(* IEC 61131-3 sources: F100R_S278_Temperville/MyController.device.xml.v3^/Plc Logic.plclogic.xml.v3^/Application.application.xml.v3^, 20 files *)

(* ---- GVL_Alarmes.gvl ---- *)
VAR_GLOBAL
	AlmMotor: ARRAY[1..25] OF BOOL;
	AlmValvAberta: ARRAY[1..12] OF BOOL;
	AlmValvFechada: ARRAY[1..12] OF BOOL;
	AlmGeral: ARRAY[1..12] OF BOOL;
	AlmEncoder: ARRAY[1..12] OF BOOL;
	AlmMotorParado: ARRAY[1..25] OF BOOL;
	xAlarmeSsrSuperiorAberto: ARRAY[1..60] OF BOOL;
	xAlarmeSsrSuperiorFechado: ARRAY[1..60] OF BOOL;
	xAlarmeSsrInferiorAberto: ARRAY[1..60] OF BOOL;
	xAlarmeSsrInferiorFechado: ARRAY[1..60] OF BOOL;
	xAlarmeResistRompidaSuperior: ARRAY[1..60] OF BOOL;
	xAlarmeResistRompidaInferior: ARRAY[1..60] OF BOOL;
	xAlarmeResistForceInferior: ARRAY[1..60] OF BOOL;
	xAlarmeResistForceSuperior: ARRAY[1..60] OF BOOL;
	xFalhaForcadaInferior: ARRAY[1..60] OF BOOL;
	xFalhaForcadaSuperior: ARRAY[1..60] OF BOOL;
	xAlarmesTestesResistenciasInferiores: ARRAY[1..60] OF BOOL;
	xAlarmesTestesResistenciasSuperiores: ARRAY[1..60] OF BOOL;
	AlmTermoparAbertoSuperior: ARRAY[1..60] OF BOOL;
	AlmTermoparAbertoInferior: ARRAY[1..60] OF BOOL;
	AlmTemperaturaExcedeuSuperior: ARRAY[1..60] OF BOOL;
	AlmTemperaturaExcedeuInferior: ARRAY[1..60] OF BOOL;
	xAlarmeSsr01ConvecEntAberto: BOOL;
	xAlarmeSsr01ConvecEntFechado: BOOL;
	xAlarmeSsr02ConvecEntAberto: BOOL;
	xAlarmeSsr02ConvecEntFechado: BOOL;
	xAlarmeSsr03ConvecEntAberto: BOOL;
	xAlarmeSsr03ConvecEntFechado: BOOL;
	xAlarmeSsr01ConvecSaiAberto: BOOL;
	xAlarmeSsr01ConvecSaiFechado: BOOL;
	xAlarmeSsr02ConvecSaiAberto: BOOL;
	xAlarmeSsr02ConvecSaiFechado: BOOL;
	xAlarmeSsr03ConvecSaiAberto: BOOL;
	xAlarmeSsr03ConvecSaiFechado: BOOL;
END_VAR

(* ---- GVL_ClpSuper.gvl ---- *)
VAR_GLOBAL
	/// LEITURA
	///Parâmetros On-line
	sEntradaNomedaReceita: STRING;
	sFornoNomedaReceita: STRING;
	sResfriamentoNomedaReceita: STRING;
	iEntradaEspessuraVidro: INT;
	iFornoEspessuraVidro: INT;
	iResfriamentoEspessuraVidro: INT;
	xEntradaReenvioRec: BOOL;
	xFornoReenvioRec: BOOL;
	xResfriamentoReenvioRec: BOOL;
	xPassagemReenvioRec: BOOL;
	rTemperaturaInferiorAtual: ARRAY[1..50] OF REAL;
	rTemperaturaSuperiorAtual: ARRAY[1..50] OF REAL;
	iTemperaturaPainel: INT;
	rMediaLogiaTempInferior: REAL;
	rMediaLogiaTempSuperior: REAL;
	rMediaLogicaTemperaturaTotal: REAL;
	iTempoDelayCargaDecorrido: INT;
	iTempoPausaRoleteDecorrido: INT;
	iTempoPausaRoleteRestante: INT;
	iTempoAquecFornoDecorrido: INT;
	iTempoAquecFornoRestante: INT;
	iTempoTrocaVelocidadeDecorrido: INT;
	///////////////////
	iTempoTrocaPosicaoDecorrido: INT;
	//////////////////
	iTempoTesteNobreak: TON;
	iTempoTesteNobreakRestante: INT;
	iTempoPausaResistInfDecorrido: INT;
	iTempoPausaResistSupDecorrido: INT;
	iTempoPausa02ResistSupDecorrido: INT;
	iTempoParaInicioPausaDecor: INT;
	iTempoConveccaoDecorrido: INT;
	iTempoResfriamentoDecorrido: INT;
	iTempoResfriamentoRestante: INT;
	iTempoTrocaEstagioDecorrido: INT;
	iTempoTrocaEstagio02Decorrido: INT;
	iAlturaAtualDuctosResfriadorInf01: INT;
	iAlturaAtualDuctosResfriadorSup01: INT;
	iAlturaAtualDuctosResfriadorInf02: INT;
	iAlturaAtualDuctosResfriadorSup02: INT;
	iAlturaAtualGuilhotina01: INT;
	iAlturaAtualGuilhotina01Sup: INT;
	iAlturaAtualGuilhotina01Inf: INT;
	iAlturaAtualGuilhotina02: INT;
	rTemperaturaPirometroInferior: REAL;
	rTemperaturaPirometroSuperior: REAL;
	iTempoStdByTemperDecorrido: INT;
	iTempoPassoSemEnerg	: INT ;
	rValorPressaoRedeMpa: REAL;
	rValorPressaoRedeBar: REAL;
	rValorPressaoRedePsi: REAL;
	///Polegada de Mercurio
	rValorPressaoRedeInHg: REAL;
	///Centimetro de Mercurio
	rValorPressaoRedeCmHg: REAL;
	///Milimetro de Mercurio
	rValorPressaoRedeMmHg: REAL;
	///Milimetro de Coluna d´agua
	rValorPressaoRedeMmCa: REAL;
	rValorPressaoMaqMpa: REAL;
	rValorPressaoMaqBar: REAL;
	rValorPressaoMaqPsi: REAL;
	///Polegada de Mercurio
	rValorPressaoMaqInHg: REAL;
	///Centimetro de Mercurio
	rValorPressaoMaqCmHg: REAL;
	///Milimetro de Mercurio
	rValorPressaoMaqMmHg: REAL;
	///Milimetro de Coluna d´agua
	rValorPressaoMaqMmCa: REAL;
	rTemperaturaTermocamera: REAL;
	rTemperaturaConveccaoEnt: REAL;
	rTemperaturaConveccaoSai: REAL;
	rValorLeituraPressaoDifusor01MBar: REAL;
	rValorLeituraPressaoDifusor01Bar: REAL;
	rValorLeituraPressaoDifusor01Psi: REAL;
	///Polegada de Mercurio
	rValorLeituraPressaoDifusor01InHg: REAL;
	///Centimetro de Mercurio
	rValorLeituraPressaoDifusor01CmHg: REAL;
	///Milimetro de Mercurio
	rValorLeituraPressaoDifusor01MmHg: REAL;
	///Milimetro de Coluna d´agua
	rValorLeituraPressaoDifusor01MmCa: REAL;
	rValorLeituraPressaoDifusor02MBar: REAL;
	rValorLeituraPressaoDifusor02Bar: REAL;
	rValorLeituraPressaoDifusor02Psi: REAL;
	///Polegada de Mercurio
	rValorLeituraPressaoDifusor02InHg: REAL;
	///Centimetro de Mercurio
	rValorLeituraPressaoDifusor02CmHg: REAL;
	///Milimetro de Mercurio
	rValorLeituraPressaoDifusor02MmHg: REAL;
	///Milimetro de Coluna d´agua
	rValorLeituraPressaoDifusor02MmCa: REAL;
	rValorVibracaoVent01: REAL;
	rValorVibracaoVent02: REAL;
	rValorVibracaoVent03: REAL;
	xResistenciaHabilitadaInferior: ARRAY[1..50] OF BOOL;
	xResistenciaHabilitadaSuperior: ARRAY[1..50] OF BOOL;
	xResistenciaHabilitada: ARRAY[1..50] OF BOOL;
	xResistenciaForcadaInferior: ARRAY[1..50] OF BOOL;
	xResistenciaForcadaSuperior: ARRAY[1..50] OF BOOL;
	xForceLigConvecEntVent: BOOL;
	xForceLigConvecSaiVent: BOOL;
	xGeralResistenciaForcada: BOOL;
	xTesteResistencias: BOOL;
	xTesteResistenciaAutomatico: BOOL;
	xTesteResistenciaManual: BOOL;
	xTesteEntradaSaidas: BOOL;
	xSelecaoTermopares: BOOL;
	xPortaEntradaFornoForce: BOOL;
	xPortaSaidaFornoForce: BOOL;
	xForceConveccao: BOOL;
	xConveccaoHabilitado: BOOL;
	xSubindoForno: BOOL;
	xDescendoForno: BOOL;
	xLigaVentiPainelManual: BOOL;
	xStdByTemperaturaHabilitado: BOOL;
	xStdByTemperaturaDesabilit: BOOL;
	xHabDesabResistConveccaoEnt: BOOL;
	xHabDesabResistConveccaoSai: BOOL;
	xAqueceRampaPatamar: BOOL;
	xAqueceReceita: BOOL;
	xAqueceRapido: BOOL;
	xAqueceLento: BOOL;
	xFimAquecimento: BOOL;
	xDuctosInf01CheckOk: BOOL;
	xDuctosSup01CheckOk: BOOL;
	xDuctosInf02CheckOk: BOOL;
	xDuctosSup02CheckOk: BOOL;
	xGuilhotina01CheckOk: BOOL;
	xGuilhotina01SupCheckOk: BOOL;
	xGuilhotina01InfCheckOk: BOOL;
	xGuilhotina02CheckOk: BOOL;
	xDuctosInf01Enable: BOOL;
	xDuctosSup01Enable: BOOL;
	xDuctosInf02Enable: BOOL;
	xDuctosSup02Enable: BOOL;
	xGuilhotina01Enable: BOOL;
	xGuilhotina01SupEnable: BOOL;
	xGuilhotina01InfEnable: BOOL;
	xGuilhotina02Enable: BOOL;
	xEnergiaOk: BOOL;
	xSemEnergia: BOOL;
	xbRestart: BOOL;
	xTesteNobreakOK: BOOL;
	xIniciaTesteNobreak: BOOL;
	xResistenciaInferiorOn: BOOL;
	xResistenciaSuperiorOn: BOOL;
	xTesteResistenciasIniciado: BOOL;
	xFimTesteResistencias: BOOL;

	xImgSetTempStandByCiclo: BOOL;

	xCircuitoEmergenciaCC : BOOL;
	xAlertaPosChCircCC	: BOOL ;
	xHabDesabCircuitoCC	: BOOL ;

	ValorAmperagemResistenciaInferior: ARRAY[1..50] OF REAL;
	ValorAmperagemResistenciaSuperior: ARRAY[1..50] OF REAL;
	xTestandoResistenciaInferior: ARRAY[1..50] OF BOOL;
	xTestandoResistenciaSuperior: ARRAY[1..50] OF BOOL;
	xFaseReleInferior: ARRAY[1..50] OF STRING;
	xFaseReleSuperior: ARRAY[1..50] OF STRING;
	iAnimaResistenciaInferior: ARRAY[1..50] OF INT;
	iAnimaResistenciaSuperior: ARRAY[1..50] OF INT;
	iAnimaResistenciaSsr01ConvecEnt: INT;
	iAnimaResistenciaSsr02ConvecEnt: INT;
	iAnimaResistenciaSsr03ConvecEnt: INT;
	iAnimaResistenciaSsr01ConvecSai: INT;
	iAnimaResistenciaSsr02ConvecSai: INT;
	iAnimaResistenciaSsr03ConvecSai: INT;
	iAnimaStatusTesteResistencias: INT;
	iAnimaTesteResistenciaInferior: ARRAY[1..50] OF INT;
	iAnimaTesteResistenciaSuperior: ARRAY[1..50] OF INT;
	iAnimaAlarmesMotores: ARRAY[1..25] OF INT;
	iAnimaAlarmesValvulas: ARRAY[1..12] OF INT;
	xTemperaturaInfeirorOk: ARRAY[1..50] OF BOOL;
	xTemperaturaSupeirorOk: ARRAY[1..50] OF BOOL;
	///Numero de cargas que sairam do resfriamento por dia
	iContaCargasResfriamento: INT;
	/// Tags Relatório de Produção
	xIniciaRelatorioProd: BOOL;
	xFinalizaRelatorioProd: BOOL;
	uNumeroCargaRel: UINT;
	rConsumoCargaRel: REAL;
	rConsumoAquecRel: REAL;
	rConsumoDiario: REAL;
	rConsumoDiarioRel: REAL;
	xGrvRelatorioEnerg: BOOL;
	iTamanhoCargaRel: INT;
	/// Tags acerta relógio
	xAcertaRelogio: BOOL;
	xRelogioAcertado: BOOL;
	/// Relatório Aquecimento
	xIniciaRelatorioAquecRampa: BOOL;
	xFinalizaRelatorioAquecRampa: BOOL;
	xIniciaRelatorioAquecRec: BOOL;
	xFinalizaRelatorioAquecRec: BOOL;
	///Tags lógica incremento
	rIncrementoTemperSup: INT;
	rIncrementoTemperInf: INT;
	rIncrementoPotenciaSup: INT;
	rIncrementoPotenciaInf: INT;
	///Tags rampas
	rTempoRampa01: REAL;
	rTempoRampa02: REAL;
	rTempoRampa03: REAL;
END_VAR

(* ---- GVL_Encoder.gvl ---- *)
VAR_GLOBAL
	dValorEncoderForno: DINT;
	dValorEncoderResfriador: DINT;
	dValorEncoderDuctosResfriadorInf01: DINT;
	dValorEncoderDuctosResfriadorSup01: DINT;
	dValorEncoderDuctosResfriadorInf02: DINT;
	dValorEncoderDuctosResfriadorSup02: DINT;
	dValorEncoderGuilhotinaResfriador01: DINT;
	dValorEncoderGuilhotinaResfriador02: DINT;

	dValorEncoderGuilhotinaResfriador01Inf: DINT;
	dValorEncoderGuilhotinaResfriador01Sup: DINT;

	xHomeEncoderForno: BOOL;
	xHomeEncoderResfriador: BOOL;
	xHomeEncoderDuctosResfriadorInf01: BOOL;
	xHomeEncoderDuctosResfriadorSup01: BOOL;
	xHomeEncoderDuctosResfriadorInf02: BOOL;
	xHomeEncoderDuctosResfriadorSup02: BOOL;
	xHomeEncoderGuilhotinaResfriador01: BOOL;
	xHomeEncoderGuilhotinaResfriador02: BOOL;
	xHomeEncoderGuilhotinaResfriador01Sup: BOOL;
	xHomeEncoderGuilhotinaResfriador01Inf: BOOL;

	xEncoderFornoOk: BOOL;
	xEncoderResfriadorOk: BOOL;
	xEncoderDuctosResfriadorInf01Ok: BOOL;
	xEncoderDuctosResfriadorSup01Ok: BOOL;
	xEncoderDuctosResfriadorInf02Ok: BOOL;
	xEncoderDuctosResfriadorSup02Ok: BOOL;
	xEncoderGuilhotinaResfriador01Ok: BOOL;
	xEncoderGuilhotinaResfriador02Ok: BOOL;
END_VAR

(* ---- GVL_Energia.gvl ---- *)
VAR_GLOBAL
	///Parametros de leituras Instantaneas Reais do PM710 para o Supervisório
	rConsumoEnergiaReal_kWh: REAL;
	rConsumoEnergiaAparente_kVAh: REAL;
	rConsumoEnergiaReativa_kVARh: REAL;
	rPotenciaTotalReal_kW: REAL;
	rPotenciaTotalAparente_kVA: REAL;
	rPotenciaTotalReativa_kVAR: REAL;
	rFatorDePotenciaTotal: REAL;
	rTensaoFFMedia_V: REAL;
	rTensaoFNMedia_V: REAL;
	rCorrenteMedia_V: REAL;
	rFrequencia_Hz: REAL;
	rDemandaTotalReal_kW: REAL;
	rDemandaTotalAparente_kVA: REAL;
	rDemandaTotalReativa_kVAR: REAL;
	rDemandaMaximaReal_kW: REAL;
	rDemandaMaximaAparente_kVA: REAL;
	rDemandaMaximaReativa_kVAR: REAL;
	rCorrenteInstantFaseA_Amp: REAL;
	rCorrenteInstantFaseB_Amp: REAL;
	rCorrenteInstantFaseC_Amp: REAL;
	rCorrenteInstantNeutro_Amp: REAL;
	rCorrenteDemandaFaseA_Amp: REAL;
	rCorrenteDemandaFaseB_Amp: REAL;
	rCorrenteDemandaFaseC_Amp: REAL;
	rCorrenteMaximaDemandaFaseA_Amp: REAL;
	rCorrenteMaximaDemandaFaseB_Amp: REAL;
	rCorrenteMaximaDemandaFaseC_Amp: REAL;
	rTensaoFaseAB_V: REAL;
	rTensaoFaseBC_V: REAL;
	rTensaoFaseAC_V: REAL;
	rTensaoFaseAN_V: REAL;
	rTensaoFaseBN_V: REAL;
	rTensaoFaseCN_V: REAL;
	rPotenciaRealFaseA_kW: REAL;
	rPotenciaRealFaseB_kW: REAL;
	rPotenciaRealFaseC_kW: REAL;
	rPotenciaAparenteFaseA_kVA: REAL;
	rPotenciaAparenteFaseB_kVA: REAL;
	rPotenciaAparenteFaseC_kVA: REAL;
	rPotenciaReativaFaseA_kVAR: REAL;
	rPotenciaReativaFaseB_kVAR: REAL;
	rPotenciaReativaFaseC_kVAR: REAL;
	rCorrenteTHDFaseA: REAL;
	rCorrenteTHDFaseB: REAL;
	rCorrenteTHDFaseC: REAL;
	rCorrenteTHDNeutro: REAL;
	rTensaoTHDFaseAN: REAL;
	rTensaoTHDFaseBN: REAL;
	rTensaoTHDFaseCN: REAL;
	rTensaoTHDFaseAB: REAL;
	rTensaoTHDFaseBC: REAL;
	rTensaoTHDFaseAC: REAL;
	/// Valores minimos
	rPotenciaTotalRealMinima_kW: REAL;
	rPotenciaTotalAparenteMinima_kVA: REAL;
	rPotenciaTotalReativaMinima_kVAR: REAL;
	rFatorDePotenciaTotalMinima: REAL;
	rFrequenciaMinima_Hz: REAL;
	rCorrenteMinimaFaseA_Amp: REAL;
	rCorrenteMinimaFaseB_Amp: REAL;
	rCorrenteMinimaFaseC_Amp: REAL;
	rCorrenteMinimaNeutro_Amp: REAL;
	rTensaoMinimaFaseAN_V: REAL;
	rTensaoMinimaFaseBN_V: REAL;
	rTensaoMinimaFaseCN_V: REAL;
	rTensaoMinimaFaseAB_V: REAL;
	rTensaoMinimaFaseBC_V: REAL;
	rTensaoMinimaFaseAC_V: REAL;
	rCorrenteTHDMinimoFaseA: REAL;
	rCorrenteTHDMinimoFaseB: REAL;
	rCorrenteTHDMinimoFaseC: REAL;
	rCorrenteTHDMinimoNeutro: REAL;
	rTensaoTHDMinimoFaseAN: REAL;
	rTensaoTHDMinimoFaseBN: REAL;
	rTensaoTHDMinimoFaseCN: REAL;
	rTensaoTHDMinimoFaseAB: REAL;
	rTensaoTHDMinimoFaseBC: REAL;
	rTensaoTHDMinimoFaseAC: REAL;
	/// Valores Maximos
	rPotenciaTotalRealMaximo_kW: REAL;
	rPotenciaTotalAparenteMaximo_kVA: REAL;
	rPotenciaTotalReativaMaximo_kVAR: REAL;
	rFatorDePotenciaTotalMaximo: REAL;
	rFrequenciaMaxima_Hz: REAL;
	rCorrenteMaximoFaseA_Amp: REAL;
	rCorrenteMaximoFaseB_Amp: REAL;
	rCorrenteMaximoFaseC_Amp: REAL;
	rCorrenteMaximoNeutro_Amp: REAL;
	rTensaoMaximoFaseAN_V: REAL;
	rTensaoMaximoFaseBN_V: REAL;
	rTensaoMaximoFaseCN_V: REAL;
	rTensaoMaximoFaseAB_V: REAL;
	rTensaoMaximoFaseBC_V: REAL;
	rTensaoMaximoFaseAC_V: REAL;
	rCorrenteTHDMaximoFaseA: REAL;
	rCorrenteTHDMaximoFaseB: REAL;
	rCorrenteTHDMaximoFaseC: REAL;
	rCorrenteTHDMaximoNeutro: REAL;
	rTensaoTHDMaximoFaseAN: REAL;
	rTensaoTHDMaximoFaseBN: REAL;
	rTensaoTHDMaximoFaseCN: REAL;
	rTensaoTHDMaximoFaseAB: REAL;
	rTensaoTHDMaximoFaseBC: REAL;
	rTensaoTHDMaximoFaseAC: REAL;
	/// // // // // // // // //
	uMesFatura: UINT;
	uAnoFatura: UINT;
	bZeraAcumulado: BOOL;
	xCmdResetGeralPm: BOOL;
	// // // // // // // // //

END_VAR

(* ---- GVL_EntradasSaidas.gvl ---- *)
VAR_GLOBAL
	///ENTRADAS LÓGICAS
	///Encoder
	InputEncoderA_MeFor: BOOL;
	InputEncoderB_MeFor: BOOL;
	InputEncoderA_MeRes: BOOL;
	InputEncoderB_MeRes: BOOL;
	InputEncoderA_DuResSup01: BOOL;
	InputEncoderB_DuResSup01: BOOL;
	InputEncoderA_DuResInf01: BOOL;
	InputEncoderB_DuResInf01: BOOL;
	InputEncoderA_DuResSup02: BOOL;
	InputEncoderB_DuResSup02: BOOL;
	InputEncoderA_DuResInf02: BOOL;
	InputEncoderB_DuResInf02: BOOL;
	InputEncoderA_GuiRes01: BOOL;
	InputEncoderB_GuiRes01: BOOL;
	InputEncoderA_GuiRes02: BOOL;
	InputEncoderB_GuiRes02: BOOL;
	dValorEncoderFornoEntrada: DINT;
	dValorEncoderResfrEntrada: DINT;
	dValorEncoderDuctosResfrSup01Entrada: DINT;
	dValorEncoderDuctosResfrInf01Entrada: DINT;
	dValorEncoderDuctosResfrSup02Entrada: DINT;
	dValorEncoderDuctosResfrInf02Entrada: DINT;
	dValorEncoderGuilhoResfr01Entrada: DINT;
	dValorEncoderGuilhoResfr02Entrada: DINT;

	dValorEncoderGuilhoResfr01SupEntrada: DINT;
	dValorEncoderGuilhoResfr01InfEntrada: DINT;

	// Segurança Motor CC

	xChCircuitoEmergenciaCC	: BOOL ;
	xChHabDesabCircuitoCC	: BOOL ;

/// Mesa de Controle
	xBtIniciaCiclo: BOOL;
	xBtFinalizaCiclo: BOOL;
	xBtCalaAlarme: BOOL;
	xBtEmergencia: BOOL;
	xChAutomaticoManual: BOOL;
	///xChStandByOperacao:BOOL;
	xBtReinicia: BOOL;
	xBt01Emergencia: BOOL;
	xBt02Emergencia: BOOL;
	xBt03Emergencia: BOOL;
	xBt04Emergencia: BOOL;
	xBt05Emergencia: BOOL;
	xBt06Emergencia: BOOL;
	xBt07Emergencia: BOOL;
	xBt08Emergencia: BOOL;
	xBt09Emergencia: BOOL;
	xBt10Emergencia: BOOL;
	xBt01CalaAlarme: BOOL;
	xBt02CalaAlarme: BOOL;
	xReleSeguranca: BOOL;
	xQgeralMotores: BOOL;
	///Mesa de Entrada
	xSensorEntrada: BOOL;
	xSensorEntrada01: BOOL;
	xSensorEntrada02: BOOL;
	xSensorEntrada03: BOOL;
	xSensorEntrada04: BOOL;
	xSensorEntrada05: BOOL;
	xSensorEntrada06: BOOL;
	xSensorEntrada07: BOOL;
	xSensorEntrada08: BOOL;
	xSensorEntrada09: BOOL;
	xSensorEntrada10: BOOL;
	xBtHabilitaCarregamento: BOOL;
	xChAvancaMesaEntrada: BOOL;
	xChRecuaMesaEntrada: BOOL;
	xBtGradeEntrada: BOOL;
	xSensorGradeEntradaUp: BOOL;
	xSensorGradeEntradaDown: BOOL;
	xMotorEntradaOn: BOOL;
	///Basculante
	xBtAvancMesaBascul: BOOL;
	xBtRecuoMesaBascul: BOOL;
	xS01PistPneumRecuado: BOOL;
	xS02PistPneumAvancad: BOOL;
	xS03PistHidraulRecuado: BOOL;
	xS04PistHidraulAvancad: BOOL;
	xS05NivelaSubida: BOOL;
	xS06NivelaDescida: BOOL;
	///Mesa do Forno
	xSensorPortaEntrada: BOOL;
	xSensorPortaEntradaAberta: BOOL;
	xSensorPortaEntradaFechada: BOOL;
	xSensorPortaSaida: BOOL;
	xSensorPortaSaidaAberta: BOOL;
	xSensorPortaSaidaFechada: BOOL;
	xFcSegCalco01: BOOL;
	xFcSegCalco02: BOOL;
	xFcSegCalco03: BOOL;
	xFcSegCalco04: BOOL;
	xFcAbertoCaixaForno: BOOL;
	xFcFechadoCaixaForno: BOOL;
	xMotorFornoOn: BOOL;

	//Ventilador Passagem
	xResetVentilador01 : BOOL;
	xRefUpVentiladorPassagem : BOOL;
	xRefDownVentiladorPassagem : BOOL;
	//Guilhotina Passagem Inferior
	xFcMaximoGuiPassagemInf : BOOL;
	xFcMinimoGuiPassagemInf : BOOL;
	//Guilhotina Passagem Superior
	xFcMaximoGuiPassagemSup : BOOL;
	xFcMinimoGuiPassagemSup : BOOL;

	///Mesa do Resfriador
	xFcLimMaxLimpaResfriador02: BOOL;
	xFcLimMinLimpaResfriador02: BOOL;
	xChAvancoLimpaResfriador02: BOOL;
	xChRecuoLimpaResfriador02: BOOL;
	xMotorResfriadorOn: BOOL;
	///Mesa de Saída
	xChAvancaMesaSaida: BOOL;
	xChRecuaMesaSaida: BOOL;
	xSensorDesligaMesaSaida: BOOL;
	xBtGradeSaida: BOOL;
	xSensorGradeSaidaUp: BOOL;
	xSensorGradeSaidaDown: BOOL;
	xMotorSaidaOn: BOOL;
	///Resfriador Inferior 01
	xSensorAbertoResfriadorInf01: BOOL;
	xSensorFechadoResfriadorInf01: BOOL;
	xSensorEncoderResfriadorInf01: BOOL;
	xChAbreDuctosResfriadorInf01: BOOL;
	xFcMinimoSegResfriadorInf01: BOOL;
	xFcMaximoSegResfriadorInf01: BOOL;
	///Resfriador Superior 01
	xSensorAbertoResfriadorSup01: BOOL;
	xSensorFechadoResfriadorSup01: BOOL;
	xSensorEncoderResfriadorSup01: BOOL;
	xChAbreDuctosResfriadorSup01: BOOL;
	xFcMinimoSegResfriadorSup01: BOOL;
	xFcMaximoSegResfriadorSup01: BOOL;
	xValvulaVeneziana: BOOL;
	xMotorResfridorSup01Abre: BOOL;
	xMotorResfridorSup01Fecha: BOOL;
	///Resfriador Inferior 02
	xSensorAbertoResfriadorInf02: BOOL;
	xSensorFechadoResfriadorInf02: BOOL;
	xSensorEncoderResfriadorInf02: BOOL;
	xChAbreDuctosResfriadorInf02: BOOL;
	xFcMinimoSegResfriadorInf02: BOOL;
	xFcMaximoSegResfriadorInf02: BOOL;
	xMotorResfridorInf02Abre: BOOL;
	xMotorResfridorInf02Fecha: BOOL;
	///Resfriador Superior 02
	xSensorAbertoResfriadorSup02: BOOL;
	xSensorFechadoResfriadorSup02: BOOL;
	xSensorEncoderResfriadorSup02: BOOL;
	xChAbreDuctosResfriadorSup02: BOOL;
	xFcMinimoSegResfriadorSup02: BOOL;
	xFcMaximoSegResfriadorSup02: BOOL;
	xMotorResfridorSup02Abre: BOOL;
	xMotorResfridorSup02Fecha: BOOL;
	///Guilhotina 01
	xSensorPositivoGuilhotina01: BOOL;
	xSensorZeroGuilhotina01: BOOL;
	xSensorNegativoGuilhotina01: BOOL;
	xSensorEncoderGuilhotina01: BOOL;
	xMotorGuilhotina01Sobe: BOOL;
	xMotorGuilhotina01Desce: BOOL;

	xSensorAbertoGuilhotina01Sup: BOOL;
	xSensorFechadoGuilhotina01Sup: BOOL;
	xMotorGuilhotina01SupAbre: BOOL;
	xMotorGuilhotina01SupFecha: BOOL;

	xSensorAbertoGuilhotina01Inf: BOOL;
	xSensorFechadoGuilhotina01Inf: BOOL;
	xMotorGuilhotina01InfAbre: BOOL;
	xMotorGuilhotina01InfFecha: BOOL;

	///Guilhotina 02
	xSensorPositivoGuilhotina02: BOOL;
	xSensorZeroGuilhotina02: BOOL;
	xSensorNegativoGuilhotina02: BOOL;
	xSensorEncoderGuilhotina02: BOOL;
	xMotorGuilhotina02Sobe: BOOL;
	xMotorGuilhotina02Desce: BOOL;
	/// Retorno Reles Estado Sólido
	xRetornoSsrInferior: ARRAY[1..60] OF BOOL;
	xRetornoSsrSuperior: ARRAY[1..60] OF BOOL;
	xRetornoSsr01ConveccaoEnt: BOOL;
	xRetornoSsr02ConveccaoEnt: BOOL;
	xRetornoSsr03ConveccaoEnt: BOOL;
	xRetornoSsr01ConveccaoSai: BOOL;
	xRetornoSsr02ConveccaoSai: BOOL;
	xRetornoSsr03ConveccaoSai: BOOL;
	/// Retorno Rele Resistências Rompidas
	xResistRompidaInferior: ARRAY[1..60] OF BOOL;
	xResistRompidaSuperior: ARRAY[1..60] OF BOOL;
	/// Amperagem Resistências
	iAmperagemInferior: ARRAY[1..60] OF UINT;
	iAmperagemSuperior: ARRAY[1..60] OF UINT;
	/// Nobreak
	xSaidaNobreakOk: BOOL;
	/// Pressostato Rede Alimnetação de Ar Comprimido
	xPressaoBaixaMediaRede: BOOL;
	xPressaoMediaAltaRede: BOOL;
	/// Disjuntores
	xDisjResistOff: BOOL;
	xDisjResistOn: BOOL;
	xDisjGeralOff: BOOL;
	xDisjGeralOn: BOOL;

	/// Entradas Fisicas
	///TM262L10MESE8T - 0.1
	xM0_1_DI0: BOOL;
	xM0_1_DI1: BOOL;
	xM0_1_DI2: BOOL;
	xM0_1_DI3: BOOL;
	///TM3XHSC202 - 0.2
	xM0_2_DI0: BOOL;
	xM0_2_DI1: BOOL;
	xM0_2_DI2: BOOL;
	xM0_2_DI3: BOOL;
	xM0_2_DI4: BOOL;
	xM0_2_DI5: BOOL;
	xM0_2_DI6: BOOL;
	xM0_2_DI7: BOOL;
	xM0_2_DI8: BOOL;
	xM0_2_DI9: BOOL;
	///TM3XHSC202 - 0.3
	xM0_3_DI0: BOOL;
	xM0_3_DI1: BOOL;
	xM0_3_DI2: BOOL;
	xM0_3_DI3: BOOL;
	xM0_3_DI4: BOOL;
	xM0_3_DI5: BOOL;
	xM0_3_DI6: BOOL;
	xM0_3_DI7: BOOL;
	xM0_3_DI8: BOOL;
	xM0_3_DI9: BOOL;

	///TM3DM24K - 0.4
	xM0_4_DI0: BOOL;
	xM0_4_DI1: BOOL;
	xM0_4_DI2: BOOL;
	xM0_4_DI3: BOOL;
	xM0_4_DI4: BOOL;
	xM0_4_DI5: BOOL;
	xM0_4_DI6: BOOL;
	xM0_4_DI7: BOOL;
	xM0_4_DI8: BOOL;
	xM0_4_DI9: BOOL;
	xM0_4_DI10: BOOL;
	xM0_4_DI11: BOOL;
	xM0_4_DI12: BOOL;
	xM0_4_DI13: BOOL;
	xM0_4_DI14: BOOL;
	xM0_4_DI15: BOOL;
	xM0_4_DI16: BOOL;
	xM0_4_DI17: BOOL;
	xM0_4_DI18: BOOL;
	xM0_4_DI19: BOOL;
	xM0_4_DI20: BOOL;
	xM0_4_DI21: BOOL;
	xM0_4_DI22: BOOL;
	xM0_4_DI23: BOOL;
	xM0_4_DI24: BOOL;
	xM0_4_DI25: BOOL;
	xM0_4_DI26: BOOL;
	xM0_4_DI27: BOOL;
	xM0_4_DI28: BOOL;
	xM0_4_DI29: BOOL;
	xM0_4_DI30: BOOL;
	xM0_4_DI31: BOOL;

	///TM3DM24R - 3.1
	xM3_1_DI0: BOOL;
	xM3_1_DI1: BOOL;
	xM3_1_DI2: BOOL;
	xM3_1_DI3: BOOL;
	xM3_1_DI4: BOOL;
	xM3_1_DI5: BOOL;
	xM3_1_DI6: BOOL;
	xM3_1_DI7: BOOL;
	xM3_1_DI8: BOOL;
	xM3_1_DI9: BOOL;
	xM3_1_DI10: BOOL;
	xM3_1_DI11: BOOL;
	xM3_1_DI12: BOOL;
	xM3_1_DI13: BOOL;
	xM3_1_DI14: BOOL;
	xM3_1_DI15: BOOL;

	///TM3DI32K - 3.2
	xM3_2_DI0: BOOL;
	xM3_2_DI1: BOOL;
	xM3_2_DI2: BOOL;
	xM3_2_DI3: BOOL;
	xM3_2_DI4: BOOL;
	xM3_2_DI5: BOOL;
	xM3_2_DI6: BOOL;
	xM3_2_DI7: BOOL;
	xM3_2_DI8: BOOL;
	xM3_2_DI9: BOOL;
	xM3_2_DI10: BOOL;
	xM3_2_DI11: BOOL;
	xM3_2_DI12: BOOL;
	xM3_2_DI13: BOOL;
	xM3_2_DI14: BOOL;
	xM3_2_DI15: BOOL;
	xM3_2_DI16: BOOL;
	xM3_2_DI17: BOOL;
	xM3_2_DI18: BOOL;
	xM3_2_DI19: BOOL;
	xM3_2_DI20: BOOL;
	xM3_2_DI21: BOOL;
	xM3_2_DI22: BOOL;
	xM3_2_DI23: BOOL;
	xM3_2_DI24: BOOL;
	xM3_2_DI25: BOOL;
	xM3_2_DI26: BOOL;
	xM3_2_DI27: BOOL;
	xM3_2_DI28: BOOL;
	xM3_2_DI29: BOOL;
	xM3_2_DI30: BOOL;
	xM3_2_DI31: BOOL;

	///TM3DI32K - 4.1
	xM4_1_DI0: BOOL;
	xM4_1_DI1: BOOL;
	xM4_1_DI2: BOOL;
	xM4_1_DI3: BOOL;
	xM4_1_DI4: BOOL;
	xM4_1_DI5: BOOL;
	xM4_1_DI6: BOOL;
	xM4_1_DI7: BOOL;
	xM4_1_DI8: BOOL;
	xM4_1_DI9: BOOL;
	xM4_1_DI10: BOOL;
	xM4_1_DI11: BOOL;
	xM4_1_DI12: BOOL;
	xM4_1_DI13: BOOL;
	xM4_1_DI14: BOOL;
	xM4_1_DI15: BOOL;
	xM4_1_DI16: BOOL;
	xM4_1_DI17: BOOL;
	xM4_1_DI18: BOOL;
	xM4_1_DI19: BOOL;
	xM4_1_DI20: BOOL;
	xM4_1_DI21: BOOL;
	xM4_1_DI22: BOOL;
	xM4_1_DI23: BOOL;
	xM4_1_DI24: BOOL;
	xM4_1_DI25: BOOL;
	xM4_1_DI26: BOOL;
	xM4_1_DI27: BOOL;
	xM4_1_DI28: BOOL;
	xM4_1_DI29: BOOL;
	xM4_1_DI30: BOOL;
	xM4_1_DI31: BOOL;

	///TM3DI32K - 4.2
	xM4_2_DI0: BOOL;
	xM4_2_DI1: BOOL;
	xM4_2_DI2: BOOL;
	xM4_2_DI3: BOOL;
	xM4_2_DI4: BOOL;
	xM4_2_DI5: BOOL;
	xM4_2_DI6: BOOL;
	xM4_2_DI7: BOOL;
	xM4_2_DI8: BOOL;
	xM4_2_DI9: BOOL;
	xM4_2_DI10: BOOL;
	xM4_2_DI11: BOOL;
	xM4_2_DI12: BOOL;
	xM4_2_DI13: BOOL;
	xM4_2_DI14: BOOL;
	xM4_2_DI15: BOOL;
	xM4_2_DI16: BOOL;
	xM4_2_DI17: BOOL;
	xM4_2_DI18: BOOL;
	xM4_2_DI19: BOOL;
	xM4_2_DI20: BOOL;
	xM4_2_DI21: BOOL;
	xM4_2_DI22: BOOL;
	xM4_2_DI23: BOOL;
	xM4_2_DI24: BOOL;
	xM4_2_DI25: BOOL;
	xM4_2_DI26: BOOL;
	xM4_2_DI27: BOOL;
	xM4_2_DI28: BOOL;
	xM4_2_DI29: BOOL;
	xM4_2_DI30: BOOL;
	xM4_2_DI31: BOOL;

	ImgTesteEntradas: ARRAY[1..168] OF BOOL;
	ImgEncoder: ARRAY[1..12] OF DINT;
	///SAÍDAS LÓGICAS
	/// Mesa de Controle
	xLedMaqEmCiclo: BOOL;
	xLedRestart: BOOL;
	xLedMaqEmEspera: BOOL;
	///Mesa de Entrada
	xValvulaGradeEntrada: BOOL;
	xLedCargaForno: BOOL;
	xMotorMesaEntradaAvanco: BOOL;
	xMotorMesaEntradaRecuo: BOOL;
	///Basculante
	xValvulaAbreBraco: BOOL;
	xValvulaFechBraco: BOOL;
	xValvulaAvancPneum: BOOL;
	xValvulaRecuaPneum: BOOL;
	xValvulaAvancHidra: BOOL;
	xValvulaRecuoHidra: BOOL;
	///Mesa do Forno
	xValvPortaEntradaForno: BOOL;
	xValvPortaSaidaForno: BOOL;
	xAbreCaixaForno: BOOL;
	xFechaCaixaForno: BOOL;
	xValvulaConveccao: BOOL;
	xDesabFalhInvMesaForno: BOOL;
	xMotorMesaFornoAvanco: BOOL;
	xMotorMesaFornoRecuo: BOOL;
	xLedMotFornoStop: BOOL;
	xValvulaScanner: BOOL;
	///Mesa do Passagem
	xMotorMesaPassAvanco: BOOL;
	xMotorMesaPassRecuo: BOOL;
	///Mesa do Resfriador
	xMotorMesaResfriadorAvanco: BOOL;
	xMotorMesaResfriadorRecuo: BOOL;
	///Mesa de Saída
	xValvulaGradeSaida: BOOL;
	xMotorMesaSaidaAvanco: BOOL;
	xMotorMesaSaidaRecuo: BOOL;
	///Resfriador
	xValvulaDamperDifusor: BOOL;
	/// Limpa Resfriador
	xAvancoLimpaResfriador02: BOOL;
	xRecuoLimpaResfriador02: BOOL;
	/// Ventilador 01
	xMotorVentilador01: BOOL;
	/// Ventilador 02
	xMotorVentilador02: BOOL;
	/// Ventilador 03
	xMotorVentilador03: BOOL;
	/// Conveccção Entrada
	xMotorConveccaoEnt: BOOL;
	/// Conveccção Saída
	xMotorConveccaoSai: BOOL;
	/// Rele Estado Sólido
	xReleSsrInferior: ARRAY[1..50] OF BOOL;
	xReleSsrSuperior: ARRAY[1..50] OF BOOL;
	xReleSsrConveccaoEnt: BOOL;
	xReleSsrConveccaoSai: BOOL;
	xBloqAbertCxFornoTemper: BOOL;
	xAlarmeLuminoso: BOOL;
	xAlarmeSonoro: BOOL;
	xVentiladoresPainel: BOOL;
	xVentiladoresSsr: BOOL;
	xMotorBombaHidraulica: BOOL;
	/// Coluna Sinalização
	xSinalSonoro: BOOL;
	xSinalLumVerd: BOOL;
	xSinalLumAmar: BOOL;
	xSinalLumVerm: BOOL;
	///Saidas Fisicas
	///TM262L10MESE8T - 0.1
	xM0_1_DQ0: BOOL;
	xM0_1_DQ1: BOOL;
	xM0_1_DQ2: BOOL;
	xM0_1_DQ3: BOOL;
	///TM3XHSC202 - 0.2
	xM0_2_DQ0: BOOL;
	xM0_2_DQ1: BOOL;
	xM0_2_DQ2: BOOL;
	xM0_2_DQ3: BOOL;
	xM0_2_DQ4: BOOL;
	xM0_2_DQ5: BOOL;
	xM0_2_DQ6: BOOL;
	xM0_2_DQ7: BOOL;
	///TM3XHSC202 - 0.3
	xM0_3_DQ0: BOOL;
	xM0_3_DQ1: BOOL;
	xM0_3_DQ2: BOOL;
	xM0_3_DQ3: BOOL;
	xM0_3_DQ4: BOOL;
	xM0_3_DQ5: BOOL;
	xM0_3_DQ6: BOOL;
	xM0_3_DQ7: BOOL;

	///TM3DM24R - 3.1
	xM3_1_DQ0: BOOL;
	xM3_1_DQ1: BOOL;
	xM3_1_DQ2: BOOL;
	xM3_1_DQ3: BOOL;
	xM3_1_DQ4: BOOL;
	xM3_1_DQ5: BOOL;
	xM3_1_DQ6: BOOL;
	xM3_1_DQ7: BOOL;

	///TM3DQ32TK - 3.3
	xM3_3_DQ0: BOOL;
	xM3_3_DQ1: BOOL;
	xM3_3_DQ2: BOOL;
	xM3_3_DQ3: BOOL;
	xM3_3_DQ4: BOOL;
	xM3_3_DQ5: BOOL;
	xM3_3_DQ6: BOOL;
	xM3_3_DQ7: BOOL;
	xM3_3_DQ8: BOOL;
	xM3_3_DQ9: BOOL;
	xM3_3_DQ10: BOOL;
	xM3_3_DQ11: BOOL;
	xM3_3_DQ12: BOOL;
	xM3_3_DQ13: BOOL;
	xM3_3_DQ14: BOOL;
	xM3_3_DQ15: BOOL;
	xM3_3_DQ16: BOOL;
	xM3_3_DQ17: BOOL;
	xM3_3_DQ18: BOOL;
	xM3_3_DQ19: BOOL;
	xM3_3_DQ20: BOOL;
	xM3_3_DQ21: BOOL;
	xM3_3_DQ22: BOOL;
	xM3_3_DQ23: BOOL;
	xM3_3_DQ24: BOOL;
	xM3_3_DQ25: BOOL;
	xM3_3_DQ26: BOOL;
	xM3_3_DQ27: BOOL;
	xM3_3_DQ28: BOOL;
	xM3_3_DQ29: BOOL;
	xM3_3_DQ30: BOOL;
	xM3_3_DQ31: BOOL;

	///TM3DQ32TK - 4.3
	xM4_3_DQ0: BOOL;
	xM4_3_DQ1: BOOL;
	xM4_3_DQ2: BOOL;
	xM4_3_DQ3: BOOL;
	xM4_3_DQ4: BOOL;
	xM4_3_DQ5: BOOL;
	xM4_3_DQ6: BOOL;
	xM4_3_DQ7: BOOL;
	xM4_3_DQ8: BOOL;
	xM4_3_DQ9: BOOL;
	xM4_3_DQ10: BOOL;
	xM4_3_DQ11: BOOL;
	xM4_3_DQ12: BOOL;
	xM4_3_DQ13: BOOL;
	xM4_3_DQ14: BOOL;
	xM4_3_DQ15: BOOL;
	xM4_3_DQ16: BOOL;
	xM4_3_DQ17: BOOL;
	xM4_3_DQ18: BOOL;
	xM4_3_DQ19: BOOL;
	xM4_3_DQ20: BOOL;
	xM4_3_DQ21: BOOL;
	xM4_3_DQ22: BOOL;
	xM4_3_DQ23: BOOL;
	xM4_3_DQ24: BOOL;
	xM4_3_DQ25: BOOL;
	xM4_3_DQ26: BOOL;
	xM4_3_DQ27: BOOL;
	xM4_3_DQ28: BOOL;
	xM4_3_DQ29: BOOL;
	xM4_3_DQ30: BOOL;
	xM4_3_DQ31: BOOL;

	///TM3DQ32TK - 4.4
	xM4_4_DQ0: BOOL;
	xM4_4_DQ1: BOOL;
	xM4_4_DQ2: BOOL;
	xM4_4_DQ3: BOOL;
	xM4_4_DQ4: BOOL;
	xM4_4_DQ5: BOOL;
	xM4_4_DQ6: BOOL;
	xM4_4_DQ7: BOOL;
	xM4_4_DQ8: BOOL;
	xM4_4_DQ9: BOOL;
	xM4_4_DQ10: BOOL;
	xM4_4_DQ11: BOOL;
	xM4_4_DQ12: BOOL;
	xM4_4_DQ13: BOOL;
	xM4_4_DQ14: BOOL;
	xM4_4_DQ15: BOOL;
	xM4_4_DQ16: BOOL;
	xM4_4_DQ17: BOOL;
	xM4_4_DQ18: BOOL;
	xM4_4_DQ19: BOOL;
	xM4_4_DQ20: BOOL;
	xM4_4_DQ21: BOOL;
	xM4_4_DQ22: BOOL;
	xM4_4_DQ23: BOOL;
	xM4_4_DQ24: BOOL;
	xM4_4_DQ25: BOOL;
	xM4_4_DQ26: BOOL;
	xM4_4_DQ27: BOOL;
	xM4_4_DQ28: BOOL;
	xM4_4_DQ29: BOOL;
	xM4_4_DQ30: BOOL;
	xM4_4_DQ31: BOOL;

	ForceTesteSaidas: ARRAY[1..124] OF BOOL;
	///ENTRADAS ANALÓGICAS
	bStatus00Mth0: BYTE;
	bStatus01Mth0: BYTE;
	bStatus00Mth1: BYTE;
	bStatus01Mth1: BYTE;
	bStatus00Mth2: BYTE;
	bStatus01Mth2: BYTE;
	bStatus00Mth3: BYTE;
	bStatus01Mth3: BYTE;
	bStatus00Mth4: BYTE;
	bStatus01Mth4: BYTE;
	bStatus00Mth5: BYTE;
	bStatus01Mth5: BYTE;
	bStatus00Mth6: BYTE;
	bStatus01Mth6: BYTE;
	bStatus00Mth7: BYTE;
	bStatus01Mth7: BYTE;
	bStatus00Mth8: BYTE;
	bStatus01Mth8: BYTE;
	bStatus00Mth9: BYTE;
	bStatus01Mth9: BYTE;
	TermoparInferior: ARRAY[1..50] OF INT;
	TermoparSuperior: ARRAY[1..50] OF INT;
	Termopar01Painel: INT;
	Termopar02Painel: INT;
	TermoparConveccaoEnt: INT;
	TermoparConveccaoSai: INT;
	/// 4-20mA
	iValorLeituraPressaoRede: INT;
	/// 4-20mA
	iValorLeituraPressaoMaq: INT;
	/// 4-20mA
	iValorTemperTermocamera: INT;
	/// Manometro Difusor
	iValorLeituraPressaoDifusor01: INT;
	iValorLeituraPressaoDifusor02: INT;
	/// Sensor de Vibração dos Ventiladores
	iValorLeituraSensorVibraV01: INT;
	iValorLeituraSensorVibraV02: INT;
	iValorLeituraSensorVibraV03: INT;

	iFrequenciaSaidaVentilador01	: INT ;

	///SAIDAS ANALÓGICAS
	iAnaFreqRefVentilador01			: INT ;

	xMotorOscilaResfr02Sup	: BOOL ;
	xMotorOscilaResfr02Inf	: BOOL ;

	xSensorOscilaResfr02Sup	: BOOL;
	xKaMotorOscilaResfr02Sup: BOOL;

	xSensorOscilaResfr02Inf	: BOOL;
	xKaMotorOscilaResfr02Inf: BOOL;
END_VAR

(* ---- GVL_Eventos.gvl ---- *)
VAR_GLOBAL
	///-------------- Disjuntores -------------
	bDisjGeralOn: BOOL;
	bDisjGeralOff: BOOL;
	bDisjResistOn: BOOL;
	bDisjResistOff: BOOL;
	///------- Comandos Mesa de Operação -------
	bMaquinaOperacaoStandby: BOOL;
	bMaquinaOperacaoHabilitada: BOOL;
	bEmergencia09On: BOOL;
	bEmergencia09Off: BOOL;
	b01ResetEmergencia: BOOL;
	///--- Comandos Mesa de Operação Manual ---
	bMaquinaEmManual: BOOL;
	bMaquinaEmAutoma: BOOL;
	bEmergencia10On: BOOL;
	bEmergencia10Off: BOOL;
	b02ResetEmergencia: BOOL;
	///------ Comandos Mesa de Entrada ------
	bEmergencia01On: BOOL;
	bEmergencia01Off: BOOL;
	bEmergencia02On: BOOL;
	bEmergencia02Off: BOOL;
	bConfirmaCarga: BOOL;
	bAvancoMeEntOn: BOOL;
	bAvancoMeEntOff: BOOL;
	bRecuoMeEntOn: BOOL;
	bRecuoMeEntOff: BOOL;
	bGradeEntradaUp: BOOL;
	bGradeEntradaDown: BOOL;
	bEmergencia03On: BOOL;
	bEmergencia03Off: BOOL;
	bEmergencia04On: BOOL;
	bEmergencia04Off: BOOL;
	///------ Comandos do Resfriamento ------
	bEmergencia05On: BOOL;
	bEmergencia05Off: BOOL;
	bAbreResfSup01: BOOL;
	bFechaResfSup01: BOOL;
	bAbreResfInf01: BOOL;
	bFechaResfInf01: BOOL;
	bAbreResfSup02: BOOL;
	bFechaResfSup02: BOOL;
	bAbreResfInf02: BOOL;
	bFechaResfInf02: BOOL;
	bEmergencia06On: BOOL;
	bEmergencia06Off: BOOL;
	bAvancoLimpVidroOn: BOOL;
	bAvancoLimpVidroOff: BOOL;
	bRecuoLimpVidroOn: BOOL;
	bRecuoLimpVidroOff: BOOL;
	///------- Comandos Mesa de Saida -------
	bEmergencia07On: BOOL;
	bEmergencia07Off: BOOL;
	bAvancoMeSaiOn: BOOL;
	bAvancoMeSaiOff: BOOL;
	bRecuoMeSaiOn: BOOL;
	bRecuoMeSaiOff: BOOL;
	bGradeSaidaUp: BOOL;
	bGradeSaidaDown: BOOL;
	bEmergencia08On: BOOL;
	bEmergencia08Off: BOOL;
	///------ Comandos do Supervisório ------
	bEnvioDeReceita: BOOL;
	bHimIniciaCiclo: BOOL;
	bHimFinalCiclo: BOOL;
	bBtSairForno: BOOL;
	bBtSairResfriamento: BOOL;
	bBtAbrePortaEntrForno: BOOL;
	bBtFechaPortaEntForno: BOOL;
	bBtAbrePortaSaidaForno: BOOL;
	bBtFechaPortaSaidForno: BOOL;
	bBtForceConveccaoOn: BOOL;
	bBtForceConveccaoOff: BOOL;
	bBtSobeGuilhtinaManual: BOOL;
	bBtDesceGuilhotinaManual: BOOL;
	bBtSobeForno: BOOL;
	bBtDesceForno: BOOL;
	bResistenciaLigada: BOOL;
	bResistenciaDesligada: BOOL;
	bTesteAutoResistencia: BOOL;
	bTesteAutoResistFim: BOOL;
	bTesteAutoResistAbort: BOOL;
	bProgrHorariaAtivada: BOOL;
	bProgrHorariaDesativada: BOOL;
	bProgrHorariaIniciadda: BOOL;
	bBtLigaAquecimentoRampa: BOOL;
	bBtLigaAquecimento: BOOL;
	bBtDesligaAquecimento: BOOL;
	bHomeDutosIniciado: BOOL;
	bHomeDutosOK: BOOL;
	bHomeGuilhotinaIniciado: BOOL;
	bHomeGuilhotinaOK: BOOL;
END_VAR

(* ---- GVL_Imagens.gvl ---- *)
VAR_GLOBAL
	ImgMotor: ARRAY[1..25] OF BOOL;
	ImgValvAberta: ARRAY[1..10] OF BOOL;
	ImgValvFechada: ARRAY[1..10] OF BOOL;
	ImgGeral: ARRAY[1..20] OF BOOL;
	ImgRetornoSsrInferior: ARRAY[1..60] OF BOOL;
	ImgRetornoSsrSuperior: ARRAY[1..60] OF BOOL;
	ImgResistenciaInferior: ARRAY[1..60] OF BOOL;
	ImgResistenciaSuperior: ARRAY[1..60] OF BOOL;
	ImgResistenciaHabilitadaInferior: ARRAY[1..60] OF BOOL;
	ImgResistenciaHabilitadaSuperior: ARRAY[1..60] OF BOOL;
END_VAR

(* ---- GVL_Interface.gvl ---- *)
VAR_GLOBAL
	xInicioPrimeiroEstagio: BOOL;
	xInicioSegundoEstagio: BOOL;
	xFimTrocaEstagiosResfriador: BOOL;
	xEspessuraVidroFino: BOOL;
	xEspessuraVidroGrosso: BOOL;
	xEspessuraVidroFinoResfriador: BOOL;
	iVelocidadeCargaMesaEntrada: INT;
	iVelocidadeCargaMesaForno: INT;
	iVelocidadeVaiVemMesaForno: INT;
	iVelocidadeDescargaMesaForno: INT;
	iVelocidadeCargaMesaPass: INT;
	iVelocidadeVaiVemMesaPass: INT;
	iVelocidadeDescargaMesaPass: INT;
	iVelocidadeCargaMesaResfriador: INT;
	iVelocidadeVaiVemMesaResfriador: INT;
	iVelocidadeDescargaMesaResfriador: INT;
	iVelociadeCargaMesadeSaida: INT;
	xBtRecAjustaAlturaDuctosInf01: BOOL;
	xBtRecAjustaAlturaDuctosSup01: BOOL;
	xBtRecAjustaAlturaDuctosInf02: BOOL;
	xBtRecAjustaAlturaDuctosSup02: BOOL;
	xBtRecAjustaGuilhotina01: BOOL;
	xBtRecAjustaGuilhotina01Sup: BOOL;
	xBtRecAjustaGuilhotina01Inf: BOOL;
	xBtRecAjustaGuilhotina02: BOOL;
	/// relógio
	/// Programação Horaria
	xDataHoraProgOk: BOOL;
	xStatusAtvProgHoraria: BOOL;
	///Aquecimento
	xIniciaAquecimentoRec: BOOL;
	xAuxiliarLigaResistenciasInferiores: BOOL;
	xAuxiliarLigaResistenciasSuperiores: BOOL;
	xCmdIniciaCiclo: BOOL;
	xCmFinalizaCiclo: BOOL;
	rDegrauSubida: REAL;
	///rSetPointTemperatura: REAL;
	xExecutaPid: BOOL;
	rSetPointTemperaturaInferior: ARRAY[1..60] OF REAL;
	rSetPointTemperaturaSuperior: ARRAY[1..60] OF REAL;
	TermoparLogicoInferior: ARRAY[1..60] OF INT;
	TermoparLogicoSuperior: ARRAY[1..60] OF INT;
	TermoparAbertoInferior: ARRAY[1..60] OF BOOL;
	TermoparAbertoSuperior: ARRAY[1..60] OF BOOL;
	TermoparAbertoLogicoInf: ARRAY[1..60] OF BOOL;
	TermoparAbertoLogicoSup: ARRAY[1..60] OF BOOL;
	Termopar01PainelAberto: BOOL;
	Termopar02PainelAberto: BOOL;
	TermoparConvecEntAberto: BOOL;
	TermoparConvecSaiAberto: BOOL;
	AlmTermoparAbertoLogicoInf: ARRAY[1..60] OF BOOL;
	AlmTermoparAbertoLogicoSup: ARRAY[1..60] OF BOOL;
	AlmTemperaturaExcedeuLogicoInf: ARRAY[1..60] OF BOOL;
	AlmTemperaturaExcedeuLogicoSup: ARRAY[1..60] OF BOOL;
	LigaInfPorAquecimentoReceita: BOOL;
	LigaSupPorAquecimentoReceita: BOOL;
	LigaInfPorAquecimentoRampa: BOOL;
	LigaSupPorAquecimentoRampa: BOOL;
	xIniciaPausaResistencias: BOOL;
	xFimTempoPausaResistInf: BOOL;
	xFimTempoPausaResistSup: BOOL;
	xFimTempoPausa02ResistSup: BOOL;
	iTemperaturaPirometroInferior: INT;
	iTemperaturaPirometroSuperior: INT;
	iTemperaturaPirometroPainel: INT;
	rSetTemperaturaInferiorGeralAux: REAL;
	rSetTemperaturaSuperiorGeralAux: REAL;
	rSetPorcentagemInferiorGeralAux: REAL;
	rSetPorcentagemSuperiorGeralAux: REAL;
	///----------- Imagens -> 03_Geral/B_Imagens---------------
	xMotorEntradaLigado: BOOL;
	xMotorFornoLigado: BOOL;
	xMotorResfriadorLigado: BOOL;
	xMotorPassagemLigado: BOOL;
	xMotorSaidaLigado: BOOL;
	xMotorDifusorInf01Ligado: BOOL;
	xMotorDifusorSup01Ligado: BOOL;
	xMotorDifusorInf02Ligado: BOOL;
	xMotorDifusorSup02Ligado: BOOL;
	xMotorGuilhotina01Ligado: BOOL;
	xMotorGuilhotina01SupLigado: BOOL;
	xMotorGuilhotina01InfLigado: BOOL;
	xMotorGuilhotina02Ligado: BOOL;
	xMotorLimpResfr02Ligado: BOOL;
	xMotorCaixaFornoLigado: BOOL;
	xMotorVentilador01Ligado: BOOL;
	xMotorVentilador02Ligado: BOOL;
	xMotorVentilador03Ligado: BOOL;
	xMotorVentilador04Ligado: BOOL;
	xMotorBombaHidrLigado: BOOL;
	xMotorVentConvecEntLigado: BOOL;
	xMotorVentConvecSaiLigado: BOOL;
	xInvMesaEntradaHabilitado: BOOL;
	xInvMesaFornoHabilitado: BOOL;
	xInvMesaResfriadorHabilitado: BOOL;
	xInvMesaSaidaHabilitado: BOOL;
	xInvDuctosInf01Habilitado: BOOL;
	xInvDuctosSup01Habilitado: BOOL;
	xInvDuctosInf02Habilitado: BOOL;
	xInvDuctosSup02Habilitado: BOOL;
	xInvGuilhotina01Habilitado: BOOL;
	xInvGuilhotina02Habilitado: BOOL;
	xInvVentilador01Habilitado: BOOL;
	xInvVentilador02Habilitado: BOOL;
	xInvVentilador03Habilitado: BOOL;
	xInvVentilador04Habilitado: BOOL;
	xInvVentConvecHabilitado: BOOL;
	xMotorMesaEntradaDirecao: BOOL;
	xMotorMesaFornoDirecao: BOOL;
	xMotorMesaResfriadorDirecao: BOOL;
	xMotorMesaSaidaDirecao: BOOL;
	xMotorDifusorInf01Direcao: BOOL;
	xMotorDifusorSup01Direcao: BOOL;
	xMotorDifusorInf02Direcao: BOOL;
	xMotorDifusorSup02Direcao: BOOL;
	xMotorGuilhotina01Direcao: BOOL;
	xMotorGuilhotina02Direcao: BOOL;
	xMotorLimpResfr02Direcao: BOOL;
	xMotorCaixaFornoDirecao: BOOL;
	///----------- Alarmes -> 03_Geral/C_Alarmes---------------
	xAlarmePortaEntradaFornoAberta: BOOL;
	xAlarmePortaEntradaFornoFechada: BOOL;
	xAlarmePortaSaidaFornoAberta: BOOL;
	xAlarmePortaSaidaFornoFechada: BOOL;
	xAlarmePortaEntradaForno: BOOL;
	xAlarmePortaSaidaForno: BOOL;
	xAlarmeValvulaGradeSaidaUp: BOOL;
	xAlarmeValvulaGradeSaidaDown: BOOL;
	xAlarmeValvulaGradeEntradaUp: BOOL;
	xAlarmeValvulaGradeEntradaDown: BOOL;
	xAlarmeValvulaGradeSaida: BOOL;
	xAlarmeValvulaGradeEntrada: BOOL;
	xAlarmePressaoArRede: BOOL;
	xAlarmePressaoArBaixaRede: BOOL;
	xAlarmePressaoArAltaRede: BOOL;
	xAlarmePressaoArRedeSom: BOOL;
	xAlarmePressaoArMaq: BOOL;
	xAlarmePressaoArBaixaMaq: BOOL;
	xAlarmePressaoArAltaMaq: BOOL;
	xAlarmePressaoArMaqSom: BOOL;
	xAlmNobreak: BOOL;
	xAlmNobreakSom: BOOL;
	xAlmDisjGeral: BOOL;
	xAlmDisjGeralSom: BOOL;
	xAlmDisjResist: BOOL;
	xAlmDisjResistSom: BOOL;
	xLimpVidroForaPosicao: BOOL;
	xLimpVidroForaPosicaoSon: BOOL;
	xAlarmeEncoderCanalA_MeForno: BOOL;
	xAlarmeEncoderCanalB_MeForno: BOOL;
	xAlarmeGeralEncoderMeForno: BOOL;
	xAlarmeSonoroEncoderMeForno: BOOL;
	xAlarmeEncoderCanalA_MeResfriador: BOOL;
	xAlarmeEncoderCanalB_MeResfriador: BOOL;
	xAlarmeGeralEncoderMeResfriador: BOOL;
	xAlarmeSonoroEncoderMeResfriador: BOOL;
	xAlarmeEncoderCanalA_DuResfriadorSup01: BOOL;
	xAlarmeEncoderCanalB_DuResfriadorSup01: BOOL;
	xAlarmeGeralEncoderDuResfriadorSup01: BOOL;
	xAlarmeSonoroEncoderDuResfriadorSup01: BOOL;
	xAlarmeEncoderCanalA_DuResfriadorInf01: BOOL;
	xAlarmeEncoderCanalB_DuResfriadorInf01: BOOL;
	xAlarmeGeralEncoderDuResfriadorInf01: BOOL;
	xAlarmeSonoroEncoderDuResfriadorInf01: BOOL;
	xAlarmeEncoderCanalA_DuResfriadorSup02: BOOL;
	xAlarmeEncoderCanalB_DuResfriadorSup02: BOOL;
	xAlarmeGeralEncoderDuResfriadorSup02: BOOL;
	xAlarmeSonoroEncoderDuResfriadorSup02: BOOL;
	xAlarmeEncoderCanalA_DuResfriadorInf02: BOOL;
	xAlarmeEncoderCanalB_DuResfriadorInf02: BOOL;
	xAlarmeGeralEncoderDuResfriadorInf02: BOOL;
	xAlarmeSonoroEncoderDuResfriadorInf02: BOOL;
	xAlarmeEncoderCanalA_GuiResfriador01: BOOL;
	xAlarmeEncoderCanalB_GuiResfriador01: BOOL;
	xAlarmeGeralEncoderGuiResfriador01: BOOL;
	xAlarmeGeralEncoderGuiResfriadorSup01: BOOL;
	xAlarmeGeralEncoderGuiResfriadorInf01: BOOL;
	xAlarmeSonoroEncoderGuiResfriador01: BOOL;
	xAlarmeEncoderCanalA_GuiResfriador02: BOOL;
	xAlarmeEncoderCanalB_GuiResfriador02: BOOL;
	xAlarmeGeralEncoderGuiResfriador02: BOOL;
	xAlarmeSonoroEncoderGuiResfriador02: BOOL;
	xAlarmeMeFornoParado: BOOL;
	xAlarmeMeFornoParadoSom: BOOL;
	xAlarmeMeResfrParado: BOOL;
	xAlarmeMeResfrParadoSom: BOOL;
	xFalhaMotorEntrada: BOOL;
	xFalhaMotorForno: BOOL;
	xFalhaMotorPassagem: BOOL;
	xFalhaMotorResfriador: BOOL;
	xFalhaMotorSaida: BOOL;
	xFalhaMotorDifusorInf01: BOOL;
	xFalhaMotorDifusorSup01: BOOL;
	xFalhaMotorDifusorInf02: BOOL;
	xFalhaMotorDifusorSup02: BOOL;
	xFalhaMotorGuilhotina01: BOOL;
	xFalhaMotorGuilhotina01Sup: BOOL;
	xFalhaMotorGuilhotina01Inf: BOOL;
	xFalhaMotorGuilhotina02: BOOL;
	xFalhaMotorLimpResfr02: BOOL;
	xFalhaMotorCaixaForno: BOOL;
	xFalhaMotorVentilador01: BOOL;
	xFalhaMotorVentilador02: BOOL;
	xFalhaMotorVentilador03: BOOL;
	xFalhaMotorVentilador04: BOOL;
	xFalhaMotorVentConvecEnt: BOOL;
	xFalhaMotorVentConvecSai: BOOL;
	xAlarmeMotorEntrada: BOOL;
	xAlarmeMotorForno: BOOL;
	xAlarmeMotorPass: BOOL;
	xAlarmeMotorResfriador: BOOL;
	xAlarmeMotorSaida: BOOL;
	xAlarmeMotorDifusorInf01: BOOL;
	xAlarmeMotorDifusorSup01: BOOL;
	xAlarmeMotorDifusorInf02: BOOL;
	xAlarmeMotorDifusorSup02: BOOL;
	xAlarmeMotorGuilhotina01: BOOL;
	xAlarmeMotorGuilhotina01Sup: BOOL;
	xAlarmeMotorGuilhotina01Inf: BOOL;
	xAlarmeMotorGuilhotina02: BOOL;
	xAlarmeMotorLimpResfr02: BOOL;
	xAlarmeMotorCaixaForno: BOOL;
	xAlarmeMotorVentilador01: BOOL;
	xAlarmeMotorVentilador02: BOOL;
	xAlarmeMotorVentilador03: BOOL;
	xAlarmeMotorVentilador04: BOOL;
	xAlarmeMotorBombaHidraulica: BOOL;
	xAlarmeMotorVentConvecEnt: BOOL;
	xAlarmeMotorVentConvecSai: BOOL;
	xAlarmeEncoderForno: BOOL;
	xAlarmeEncoderResfriador: BOOL;
	xAlarmeEncoderDuctosResf: BOOL;
	xAlarmeEncoderGuilhotina: BOOL;
	xAlarmesResistenciasGeralInferior: ARRAY[1..60] OF BOOL;
	xAlarmesResistenciasGeralSuperior: ARRAY[1..60] OF BOOL;
	xAlarmesResistenciasGeralInferiorSon: ARRAY[1..60] OF BOOL;
	xAlarmesResistenciasGeralSuperiorSon: ARRAY[1..60] OF BOOL;
	xTesteResistenciaInferiorOk: ARRAY[1..60] OF BOOL;
	xTesteResistenciaSuperiorOk: ARRAY[1..60] OF BOOL;
	xTesteResistenciaInferiorFlh: ARRAY[1..60] OF BOOL;
	xTesteResistenciaSuperiorFlh: ARRAY[1..60] OF BOOL;
	xAlarmeSsrConvecEntAberto: BOOL;
	xAlarmeSsrConvecEntFechado: BOOL;
	xAlarmeSsrConvecSaiAberto: BOOL;
	xAlarmeSsrConvecSaiFechado: BOOL;
	xAlarmesTermopares: BOOL;
	xAlarmesTermoparesSon: BOOL;
	xAlmTermoparAbertoConvecEntSin : BOOL;
	xAlmTermoparAbertoConvecEntSon	: BOOL;
	xAlmTemperExcedeuConvecEntSin	: BOOL ;
	xAlmTemperExcedeuConvecEntSon	: BOOL;
	xAlmTermoparAbertoConvecSaiSin : BOOL;
	xAlmTermoparAbertoConvecSaiSon	: BOOL;
	xAlmTemperExcedeuConvecSaiSin	: BOOL ;
	xAlmTemperExcedeuConvecSaiSon	: BOOL;
	xAlarmesSSr: BOOL;
	xAlarmesSSrSon: BOOL;
	xAlarmesMotores: BOOL;
	xAlarmesMotoresSon: BOOL;
	xAlmSomSemEnergia: BOOL;
	wErroMotorId: ARRAY[1..60] OF WORD;
	bResetAlmGeral: BOOL;
	xBotaoResetaDrives: BOOL;
	xPause: BOOL;
	xRestart: BOOL;
	xReceitaEnviadaEventos: BOOL;
	xSairResfriamentoEventos: BOOL;
	xBtLigaResRampa: BOOL;
	xBtLigaResCiclo: BOOL;
	xBtDeslResCiclo: BOOL;

	xAlarmeSsrConvecEntSin	: BOOL;
	xAlarmeSsrConvecEntSon	: BOOL ;
	xAlarmeSsrConvecSaiSin	: BOOL;
	xAlarmeSsrConvecSaiSon	: BOOL ;
	/// Teste de Resistências
	xExecutandoTesteResistencias: BOOL;
	xPausaEmergencia: BOOL;
	xPausaEmergenciaTof: BOOL;
	///MesaEntrada
	xIniciaCargaMesaEntrada: BOOL;
	xCargaFornoEmAutomatico: BOOL;
	xCarregamentoHabilitado: BOOL;
	/// MesaForno
	xIniciaCargaForno: BOOL;
	xRecargaForno: BOOL;
	xDelayCargaForno: BOOL;
	xPortaEntradaForno: BOOL;
	xPortaSaidaForno: BOOL;
	xAvancMesaForno: BOOL;
	xRecuaMesaResfriador: BOOL;
	xAvancoMesaForno: BOOL;
	xRecuoMesaForno: BOOL;
	xLigaConveccaoForno: BOOL;
	xValvulaConveccaoLigada: BOOL;
	xSairForno: BOOL;
	xFornoComCarga: BOOL;
	xFornoEmCicloComCarga: BOOL;
	xPausaHabilitaTesteEncoder: BOOL;
	iVelocidadeMesaForno: INT;
	xExecutaMovMesaForno: BOOL;
	McMoveVelocityMesaFornoBusy: BOOL;
	xDesligaMotorFornoTempBaixa: BOOL;
	xTempoPausaRoletesOn: BOOL;
	xLedStart: BOOL;
	xAutoResetMotorForno: BOOL;
	// Mesa Passagem
	xLigaCargaPassagem: BOOL;
	xAvancoMesaPassagem: BOOL;
	xRecuoMesaPassagem: BOOL;
	xIniciaCargaPassagem: BOOL;
	///MesaResfriador
	xCancelaCargaResfriamento: BOOL;
	xLigaCargaResfriador: BOOL;
	xIniciaCargaResfriador: BOOL;
	xDesceGradeMesaSaida: BOOL;
	xAvancandMesaResfriador: BOOL;
	xRecuandoMesaResfriador: BOOL;
	xPulsoTrocaParamResfriador: BOOL;
	xSomDescarga: BOOL;
	xDesabJogMesaSaida: BOOL;
	xAbreVenezVentPass: BOOL;
	xFechVenezVentPass: BOOL;
	xPassandoTempera: BOOL;
	xAvancoMesaResfriador: BOOL;
	xRecuoMesaResfriador: BOOL;
	///Dutos Resfriador Inferior 01
	xDuctosInf01EmHome: BOOL;
	xDuctosInf01EmAjuste: BOOL;
	xAjusteAlturaDuctosInf01OK: BOOL;
	xLigaSegEstagDuctosInf01: BOOL;
	xLigaTerEstagDuctosInf01: BOOL;
	///Dutos Resfriador Superior 01
	xDuctosSup01EmHome: BOOL;
	xDuctosSup01EmAjuste: BOOL;
	xAjusteAlturaDuctosSup01OK: BOOL;
	xLigaSegEstagDuctosSup01: BOOL;
	xLigaTerEstagDuctosSup01: BOOL;
	xPausaMesaResfrimento: BOOL;
	///Dutos Resfriador Inferior 02
	xDuctosInf02EmHome: BOOL;
	xDuctosInf02EmAjuste: BOOL;
	xAjusteAlturaDuctosInf02OK: BOOL;
	xLigaSegEstagDuctosInf02: BOOL;
	xLigaTerEstagDuctosInf02: BOOL;
	///Dutos Resfriador Superior 02
	xDuctosSup02EmHome: BOOL;
	xDuctosSup02EmAjuste: BOOL;
	xAjusteAlturaDuctosSup02OK: BOOL;
	xLigaSegEstagDuctosSup02: BOOL;
	xLigaTerEstagDuctosSup02: BOOL;
	xDesceAutoFimCiclo: BOOL;
	xPausaResfrChAbreSupAcionanda: BOOL;
	/// Guilhotina 01
	xGuilhotina01EmHome: BOOL;
	xGuilhotina01EmAjuste: BOOL;
	xAjusteAlturaGuilhotina01OK: BOOL;
	/// Guilhotina 01 Superior
	xGuilhotina01SupEmHome: BOOL;
	xGuilhotina01SupEmAjuste: BOOL;
	xAjusteAlturaGuilhotina01SupOK: BOOL;
	/// Guilhotina 01 Inferior
	xGuilhotina01InfEmHome: BOOL;
	xGuilhotina01InfEmAjuste: BOOL;
	xAjusteAlturaGuilhotina01InfOK: BOOL;
	/// Guilhotina 02
	xGuilhotina02EmHome: BOOL;
	xGuilhotina02EmAjuste: BOOL;
	xAjusteAlturaGuilhotina02OK: BOOL;
	/// Ventilador 01
	xDesligaVentilador01: BOOL;
	xPrimeiroEstagioVentilador01: BOOL;
	xSegundoEstagioVentilador01: BOOL;
	xTerceiroEstagioVentilador01: BOOL;
	xVelocidadeVentilador01Ok: BOOL;
	xLigaVent01FimForno: BOOL;
	xDesligaFimVentilador01: BOOL;
	xFechaVenezVentPassV01: BOOL;
	iVelocidadeStbVent01Pass: INT;
	/// Ventilador 02
	xDesligaVentilador02: BOOL;
	xPrimeiroEstagioVentilador02: BOOL;
	xSegundoEstagioVentilador02: BOOL;
	xTerceiroEstagioVentilador02: BOOL;
	xVelocidadeVentilador02Ok: BOOL;
	xLigaVent02FimForno: BOOL;
	xDesligaFimVentilador02: BOOL;
	xFechaVenezVentPassV02: BOOL;
	iVelocidadeStbVent02Pass: INT;
	/// Ventilador 03
	xDesligaVentilador03: BOOL;
	xPrimeiroEstagioVentilador03: BOOL;
	xSegundoEstagioVentilador03: BOOL;
	xTerceiroEstagioVentilador03: BOOL;
	xVelocidadeVentilador03Ok: BOOL;
	xLigaVent03FimForno: BOOL;
	xDesligaFimVentilador03: BOOL;
	/// Ventilador 04
	xDesligaVentilador04: BOOL;
	xPrimeiroEstagioVentilador04: BOOL;
	xSegundoEstagioVentilador04: BOOL;
	xTerceiroEstagioVentilador04: BOOL;
	xVelocidadeVentilador04Ok: BOOL;
	xLigaVent04FimForno: BOOL;
	xDesligaFimVentilador04: BOOL;
	xBufferValvulaDamperDifusor: BOOL;
	/// Caixa do Forno
	xAlertaSomCxForno: BOOL;
	/// Resistencia
	xSaidaReleRampaPatamarInf: ARRAY[1..60] OF BOOL;
	xSaidaReleRampaPatamarSup: ARRAY[1..60] OF BOOL;
	xResistenciaInferior: ARRAY[1..60] OF BOOL;
	xResistenciaSuperior: ARRAY[1..60] OF BOOL;
	xResetErro: BOOL;
	/// Resistencias Convecção
	xRetornoSsrConveccaoEnt: BOOL;
	xRetornoSsrConveccaoSai: BOOL;
	///---------------------------------
	xSetTempStandyByInicio: BOOL;
	xStartCargaForno: BOOL;
	xFimDescForIniStdBy: BOOL;
	///Nobreak
	xStatusNobreak: BOOL;
	xNobreakDesabilitado: BOOL;
	/// Energia
	xSomSemEnergia: BOOL;
	dSomaReceitaClp: DINT;
	xBloqueioCargaEnvioRec: BOOL;
	xTempoDesligaResistQ: BOOL;
	/// Encoder
	///Mesa Forno
	xRunEncoMForno: BOOL;
	xErrEncoMForno: BOOL;
	xPresetEncoMForno: BOOL;
	///Mesa Resfriamento
	xRunEncoMResfr: BOOL;
	xErrEncoMResfr: BOOL;
	xPresetEncoMResfr: BOOL;
	/// Resfriador - Dutos Superior
	xRunEncoResfrSup02: BOOL;
	xErrEncoResfrSup02: BOOL;
	xPresetEncoResfrSup02: BOOL;
	/// Resfriador - Dutos Inferior
	xRunEncoResfrInf02: BOOL;
	xErrEncoResfrInf02: BOOL;
	xPresetEncoResfrInf02: BOOL;
	/// Guilhotina Resfriador
	xRunEncoGuilhotina02: BOOL;
	xErrEncoGuilhortina02: BOOL;
	xPresetEncoGuilhotina02: BOOL;
	/// Mesa Passagem
	xRunEncoMPassagem : BOOL;
	xErrEncoMPassagem : BOOL;
	xPressetEncoMPassagem : BOOL;
	/// Passagem - Dutos Superior
	xRunEncoResfrSup01: BOOL;
	xErrEncoResfrSup01: BOOL;
	xPresetEncoResfrSup01: BOOL;
	/// Passagem - Dutos Inferior
	xRunEncoResfrInf01: BOOL;
	xErrEncoResfrInf01: BOOL;
	xPresetEncoResfrInf01: BOOL;
	/// Guilhotina Passagem
	xRunEncoGuilhotina01: BOOL;
	xErrEncoGuilhortina01: BOOL;
	xPresetEncoGuilhotina01: BOOL;
	/// Passagem - Guilhotina Superior
	xRunEncoGuilhotina01Sup: BOOL;
	xErrEncoGuilhortina01Sup: BOOL;
	xPresetEncoGuilhotina01Sup: BOOL;
	/// Passagem - Guilhotina Inferior
	xRunEncoGuilhotina01Inf: BOOL;
	xErrEncoGuilhortina01Inf: BOOL;
	xPresetEncoGuilhotina01Inf: BOOL;

	xPulsoOperacaoManual: BOOL;
	xPulsoOperacaoAutoma: BOOL;
	xTonOperacaoManual: BOOL;
	xTonOperacaoAutoma: BOOL;
	xTofOperacaoManual: BOOL;
	xTofOperacaoAutoma: BOOL;

	iNumResistencias:INT;

	xResetPid:BOOL;

	xAutoHomeResfInf02	: BOOL ;
	xAutoHomeResfSup02	: BOOL ;
	xAutoHomeGuilho01	: BOOL ;
	xAutoHomeGuilho02	: BOOL ;

		xForceDut : BOOL ;

			xAlarmeMotorOscilaSup02: BOOL ;
	xAlarmeMotorOscilaInf02: BOOL;

END_VAR

(* ---- GVL_InterfaceEnergia.gvl ---- *)
VAR_GLOBAL
	/// 3000
	wCorrenteFaseA_MW0 AT %MW0: WORD;
	/// 2999
	wCorrenteFaseA_MW1 AT %MW1: WORD;
	/// 3002
	wCorrenteFaseB_MW0 AT %MW4: WORD;
	/// 3001
	wCorrenteFaseB_MW1 AT %MW5: WORD;
	/// 3004
	wCorrenteFaseC_MW0 AT %MW8: WORD;
	/// 3003
	wCorrenteFaseC_MW1 AT %MW9: WORD;
	/// 3006
	wCorrenteNeutro_MW0 AT %MW12: WORD;
	/// 3005
	wCorrenteNeutro_MW1 AT %MW13: WORD;
	/// 3008
	wCorrenteG_MW0 AT %MW16: WORD;
	/// 3007
	wCorrenteG_MW1 AT %MW17: WORD;
	/// 3010
	wCorrenteAvg_MW0 AT %MW20: WORD;
	/// 3009
	wCorrenteAvg_MW1 AT %MW21: WORD;
	/// 3020
	wTensaoAB_MW0 AT %MW40: WORD;
	/// 3019
	wTensaoAB_MW1 AT %MW41: WORD;
	/// 3022
	wTensaoBC_MW0 AT %MW44: WORD;
	/// 3021
	wTensaoBC_MW1 AT %MW45: WORD;
	/// 3024
	wTensaoCA_MW0 AT %MW48: WORD;
	/// 3023
	wTensaoCA_MW1 AT %MW49: WORD;
	/// 3026
	wTensaoAvgL_MW0 AT %MW52: WORD;
	/// 3025
	wTensaoAvgL_MW1 AT %MW53: WORD;
	/// 3028
	wTensaoAN_MW0 AT %MW56: WORD;
	/// 3027
	wTensaoAN_MW1 AT %MW57: WORD;
	/// 3030
	wTensaoBN_MW0 AT %MW60: WORD;
	/// 3029
	wTensaoBN_MW1 AT %MW61: WORD;
	/// 3032
	wTensaoCN_MW0 AT %MW64: WORD;
	/// 3031
	wTensaoCN_MW1 AT %MW65: WORD;
	/// 3036
	wTensaoAvgN_MW0 AT %MW72: WORD;
	/// 3035
	wTensaoAvgN_MW1 AT %MW73: WORD;
	///3060
	wPotenciaAtivaTotal_MW0 AT %MW120: WORD;
	///3059
	wPotenciaAtivaTotal_MW1 AT %MW121: WORD;
	///3084
	wFatorPotenciaTotal_MW0 AT %MW168: WORD;
	///3083
	wFatorPotenciaTotal_MW1 AT %MW169: WORD;
	///3110
	wFrequencia_MW0 AT %MW220: WORD;
	///3109
	wFrequencia_MW1 AT %MW221: WORD;
	///3763
	wUltimaDemanda_MW0 AT %MW300: WORD;
	///3762
	wUltimaDemanda_MW1 AT %MW301: WORD;
	///3765
	wAtualDemanda_MW0 AT %MW304: WORD;
	///3764
	wAtualDemanda_MW1 AT %MW305: WORD;
	///3767
	wPrevisaoDemanda_MW0 AT %MW308: WORD;
	///3766
	wPrevisaoDemanda_MW1 AT %MW309: WORD;
	///3769
	wPicoDemanda_MW0 AT %MW312: WORD;
	///3768
	wPicoDemanda_MW1 AT %MW313: WORD;
	///3204
	wEnergiaAtivaAcumulada_MW0_High AT %MW500: WORD;
	///3203
	wEnergiaAtivaAcumulada_MW1_High AT %MW501: WORD;
	///3206
	wEnergiaAtivaAcumulada_MW0_Low AT %MW504: WORD;
	///3205
	wEnergiaAtivaAcumulada_MW1_Low AT %MW505: WORD;
	///3220
	wEnergiaReativaAcumulada_MW0_High AT %MW510: WORD;
	///3219
	wEnergiaReativaAcumulada_MW1_High AT %MW511: WORD;
	///3222
	wEnergiaReativaAcumulada_MW0_Low AT %MW514: WORD;
	///3221
	wEnergiaReativaAcumulada_MW1_Low AT %MW515: WORD;
	///3236
	wEnergiaAparenteAcumulada_MW0_High AT %MW520: WORD;
	///3235
	wEnergiaAparenteAcumulada_MW1_High AT %MW521: WORD;
	///3238
	wEnergiaAparenteAcumulada_MW0_Low AT %MW524: WORD;
	///3237
	wEnergiaAparenteAcumulada_MW1_Low AT %MW525: WORD;
	/// Memórias Float
	fCorrenteFaseA AT %MD0: REAL;
	fCorrenteFaseB AT %MD2: REAL;
	fCorrenteFaseC AT %MD4: REAL;
	fCorrenteNeutro AT %MD6: REAL;
	fCorrenteG AT %MD8: REAL;
	fCorrenteAvg AT %MD10: REAL;
	fTensaoAB AT %MD20: REAL;
	fTensaoBC AT %MD22: REAL;
	fTensaoCA AT %MD24: REAL;
	fTensaoAvgLL AT %MD26: REAL;
	fTensaoAN AT %MD28: REAL;
	fTensaoBN AT %MD30: REAL;
	fTensaoCN AT %MD32: REAL;
	fTensaoAvgLN AT %MD36: REAL;
	fPotenciaAtivaTotal AT %MD60: REAL;
	fFatorPotenciaTotal AT %MD84: REAL;
	fFrequencia AT %MD110: REAL;
	fUltimaDemanda AT %MD150: REAL;
	fAtualDemanda AT %MD152: REAL;
	fPrevisaoDemanda AT %MD154: REAL;
	fPicoDemanda AT %MD156: REAL;
	///3204
	dEnergiaAtivaAcumulada_D_High AT %MD250: DINT;
	///3206
	dEnergiaAtivaAcumulada_D_Low AT %MD252: DINT;
	///3220
	dEnergiaReativaAcumulada_D_High AT %MD255: DINT;
	///3222
	dEnergiaReativaAcumulada_D_Low AT %MD257: DINT;
	///3236
	dEnergiaAparenteAcumulada_D_High AT %MD260: DINT;
	///3238
	dEnergiaAparenteAcumulada_D_Low AT %MD262: DINT;
	fEnergiaAtivaAcumulada: REAL;
	fEnergiaReativaAcumulada: REAL;
	fEnergiaAparenteAcumulada: REAL;
	/// Valores Máximos
	fCorrenteMaximaFaseA: REAL;
	fCorrenteMaximaFaseB: REAL;
	fCorrenteMaximaFaseC: REAL;
	fCorrenteMaximaNeutro: REAL;
	fCorrenteMaximaG: REAL;
	fCorrenteMaximaAvg: REAL;
	fTensaoMaximaAB: REAL;
	fTensaoMaximaBC: REAL;
	fTensaoMaximaCA: REAL;
	fTensaoMaximaAvgL: REAL;
	fTensaoMaximaAN: REAL;
	fTensaoMaximaBN: REAL;
	fTensaoMaximaCN: REAL;
	fTensaoMaximaAvgN: REAL;
	fPotenciaAtivaTotalMaxima: REAL;
END_VAR

(* ---- GVL_InterfacePid.gvl ---- *)
VAR_GLOBAL
	Index: INT;
	xAlternaSetor: BOOL;
	TB01: blink;
	/// Resistências Inferiores
	ControleInferiorSetor01: PidPwm_ONOFF;
	ControleInferiorSetor02: PidPwm_ONOFF;
	ControleInferiorSetor03: PidPwm_ONOFF;
	ControleInferiorSetor04: PidPwm_ONOFF;
	ControleInferiorSetor05: PidPwm_ONOFF;
	ControleInferiorSetor06: PidPwm_ONOFF;
	ControleInferiorSetor07: PidPwm_ONOFF;
	ControleInferiorSetor08: PidPwm_ONOFF;
	ControleInferiorSetor09: PidPwm_ONOFF;
	ControleInferiorSetor10: PidPwm_ONOFF;
	ControleInferiorSetor11: PidPwm_ONOFF;
	ControleInferiorSetor12: PidPwm_ONOFF;
	ControleInferiorSetor13: PidPwm_ONOFF;
	ControleInferiorSetor14: PidPwm_ONOFF;
	ControleInferiorSetor15: PidPwm_ONOFF;
	ControleInferiorSetor16: PidPwm_ONOFF;
	ControleInferiorSetor17: PidPwm_ONOFF;
	ControleInferiorSetor18: PidPwm_ONOFF;
	ControleInferiorSetor19: PidPwm_ONOFF;
	ControleInferiorSetor20: PidPwm_ONOFF;
	ControleInferiorSetor21: PidPwm_ONOFF;
	ControleInferiorSetor22: PidPwm_ONOFF;
	ControleInferiorSetor23: PidPwm_ONOFF;
	ControleInferiorSetor24: PidPwm_ONOFF;
	ControleInferiorSetor25: PidPwm_ONOFF;
	ControleInferiorSetor26: PidPwm_ONOFF;
	ControleInferiorSetor27: PidPwm_ONOFF;
	ControleInferiorSetor28: PidPwm_ONOFF;
	ControleInferiorSetor29: PidPwm_ONOFF;
	ControleInferiorSetor30: PidPwm_ONOFF;
	ControleInferiorSetor31: PidPwm_ONOFF;
	ControleInferiorSetor32: PidPwm_ONOFF;
	ControleInferiorSetor33: PidPwm_ONOFF;
	ControleInferiorSetor34: PidPwm_ONOFF;
	ControleInferiorSetor35: PidPwm_ONOFF;
	ControleInferiorSetor36: PidPwm_ONOFF;
	ControleInferiorSetor37: PidPwm_ONOFF;
	ControleInferiorSetor38: PidPwm_ONOFF;
	ControleInferiorSetor39: PidPwm_ONOFF;
	ControleInferiorSetor40: PidPwm_ONOFF;
	ControleInferiorSetor41: PidPwm_ONOFF;
	ControleInferiorSetor42: PidPwm_ONOFF;
	ControleInferiorSetor43: PidPwm_ONOFF;
	ControleInferiorSetor44: PidPwm_ONOFF;
	ControleInferiorSetor45: PidPwm_ONOFF;
	ControleInferiorSetor46: PidPwm_ONOFF;
	ControleInferiorSetor47: PidPwm_ONOFF;
	ControleInferiorSetor48: PidPwm_ONOFF;
	ControleInferiorSetor49: PidPwm_ONOFF;
	ControleInferiorSetor50: PidPwm_ONOFF;

	rTermoparInferiorLeitura: ARRAY[1..60] OF REAL;
	rTermoparInferiorControle: ARRAY[1..60] OF REAL;
	rTemperaturaInferiorSetor: ARRAY[1..60] OF REAL;
	xRrsInferiorSetor: ARRAY[1..60] OF BOOL;
	xLigaDeslResInferiores: BOOL;
	xLigaDesligaInfG01: BOOL;
	xLigaDesligaInfG02: BOOL;
	/// Resistências Superiores
	ControleSuperiorSetor01: PidPwm_ONOFF;
	ControleSuperiorSetor02: PidPwm_ONOFF;
	ControleSuperiorSetor03: PidPwm_ONOFF;
	ControleSuperiorSetor04: PidPwm_ONOFF;
	ControleSuperiorSetor05: PidPwm_ONOFF;
	ControleSuperiorSetor06: PidPwm_ONOFF;
	ControleSuperiorSetor07: PidPwm_ONOFF;
	ControleSuperiorSetor08: PidPwm_ONOFF;
	ControleSuperiorSetor09: PidPwm_ONOFF;
	ControleSuperiorSetor10: PidPwm_ONOFF;
	ControleSuperiorSetor11: PidPwm_ONOFF;
	ControleSuperiorSetor12: PidPwm_ONOFF;
	ControleSuperiorSetor13: PidPwm_ONOFF;
	ControleSuperiorSetor14: PidPwm_ONOFF;
	ControleSuperiorSetor15: PidPwm_ONOFF;
	ControleSuperiorSetor16: PidPwm_ONOFF;
	ControleSuperiorSetor17: PidPwm_ONOFF;
	ControleSuperiorSetor18: PidPwm_ONOFF;
	ControleSuperiorSetor19: PidPwm_ONOFF;
	ControleSuperiorSetor20: PidPwm_ONOFF;
	ControleSuperiorSetor21: PidPwm_ONOFF;
	ControleSuperiorSetor22: PidPwm_ONOFF;
	ControleSuperiorSetor23: PidPwm_ONOFF;
	ControleSuperiorSetor24: PidPwm_ONOFF;
	ControleSuperiorSetor25: PidPwm_ONOFF;
	ControleSuperiorSetor26: PidPwm_ONOFF;
	ControleSuperiorSetor27: PidPwm_ONOFF;
	ControleSuperiorSetor28: PidPwm_ONOFF;
	ControleSuperiorSetor29: PidPwm_ONOFF;
	ControleSuperiorSetor30: PidPwm_ONOFF;
	ControleSuperiorSetor31: PidPwm_ONOFF;
	ControleSuperiorSetor32: PidPwm_ONOFF;
	ControleSuperiorSetor33: PidPwm_ONOFF;
	ControleSuperiorSetor34: PidPwm_ONOFF;
	ControleSuperiorSetor35: PidPwm_ONOFF;
	ControleSuperiorSetor36: PidPwm_ONOFF;
	ControleSuperiorSetor37: PidPwm_ONOFF;
	ControleSuperiorSetor38: PidPwm_ONOFF;
	ControleSuperiorSetor39: PidPwm_ONOFF;
	ControleSuperiorSetor40: PidPwm_ONOFF;
	ControleSuperiorSetor41: PidPwm_ONOFF;
	ControleSuperiorSetor42: PidPwm_ONOFF;
	ControleSuperiorSetor43: PidPwm_ONOFF;
	ControleSuperiorSetor44: PidPwm_ONOFF;
	ControleSuperiorSetor45: PidPwm_ONOFF;
	ControleSuperiorSetor46: PidPwm_ONOFF;
	ControleSuperiorSetor47: PidPwm_ONOFF;
	ControleSuperiorSetor48: PidPwm_ONOFF;
	ControleSuperiorSetor49: PidPwm_ONOFF;
	ControleSuperiorSetor50: PidPwm_ONOFF;

	rTermoparSuperiorLeitura: ARRAY[1..60] OF REAL;
	rTermoparSuperiorControle: ARRAY[1..60] OF REAL;
	rTemperaturaSuperiorSetor: ARRAY[1..60] OF REAL;
	xRrsSuperiorSetor: ARRAY[1..60] OF BOOL;
	xLigaDeslResSuperiores: BOOL;
	xLigaDesligaSupG01: BOOL;
	xLigaDesligaSupG02: BOOL;
	xResistenciaInferiorPausa: BOOL;
	xResistenciaSuperiorPausa01: BOOL;
	xResistenciaSuperiorPausa02: BOOL;
	xLigaResistenciaInferior: BOOL;
	xLigaResistenciaSuperior: BOOL;
	TemporizaPausaResistInferior: Temporizador;
	TemporizaPausaResistSuperior: Temporizador;
	TempoInicioPausa02ResistSuperior: TON;
	TemporizaPausa02ResistSuperior: Temporizador;
	xIniciaPausaResistInf: BOOL;
	xIniciaPausaResistSup: BOOL;
	xIniciaTempoPausaResistSup: BOOL;
	xIniciaPausa02ResistSup: BOOL;
	xHabilitaBlocosControle: BOOL;
	xHabilitaBlocosControleInferior: BOOL;
	xHabilitaBlocosControleSuperior: BOOL;
	///-------- Teste PID ------------
	rPidSaida: REAL;
	rPwmEntrada: REAL;
	PID: FB_PID;
	PWM: FB_PWM;
	xHabilitaControle: BOOL;
	rGanhoPorporcionaKp: REAL;
	rGanhoIntegralKi: REAL;
	rGanhoDerivativoKd: REAL;

	xReleSsrSuperiorRampa74: BOOL;
END_VAR

(* ---- GVL_Inversores.gvl ---- *)
VAR_GLOBAL
	InversorMesaEntrada: Inversor;
	InversorMesaForno: Inversor;
	InversorMesaPass: Inversor;
	InversorMesaResfri: Inversor;
	InversorMesaSaida: Inversor;
	InversorResfSup01: Inversor;
	InversorResfInf01: Inversor;
	InversorResfSup02: Inversor;
	InversorResfInf02: Inversor;
	InversorGuilhot01: Inversor;
	InversorGuilhot02: Inversor;
	InversorVentila01: Inversor;
	InversorVentila02: Inversor;
	InversorVentila03: Inversor;
	InversorVentila04: Inversor;
	InversorConvecEnt: Inversor;
	InversorConvecSai: Inversor;
	InversorSobeDesceForno : Inversor;
	InversorGuilhot01Sup: Inversor;
	InversorGuilhot01Inf: Inversor;
END_VAR

(* ---- GVL_Motores.gvl ---- *)
VAR_GLOBAL
	uAmperagemMotorMesaEntrada: UINT;
	iFrequenciaMotorMesaEntrada: INT;
	uAmperagemMotorMesaForno: UINT;
	iFrequenciaMotorMesaForno: INT;
	uAmperagemMotorMesaPassagem: UINT;
	iFrequenciaMotorMesaPassagem: INT;
	uAmperagemMotorMesaResfriamento: UINT;
	iFrequenciaMotorMesaResfriamento: INT;
	uAmperagemMotorMesaSaida: UINT;
	iFrequenciaMotorMesaSaida: INT;
	uAmperagemMotorDutosResfriadorInf01: UINT;
	iFrequenciaMotorDutosResfriadorInf01: INT;
	uAmperagemMotorDutosResfriadorSup01: UINT;
	iFrequenciaMotorDutosResfriadorSup01: INT;
	uAmperagemMotorDutosResfriadorInf02: UINT;
	iFrequenciaMotorDutosResfriadorInf02: INT;
	uAmperagemMotorDutosResfriadorSup02: UINT;
	iFrequenciaMotorDutosResfriadorSup02: INT;
	uAmperagemMotorGuilhotina01: UINT;
	iFrequenciaMotorGuilhotina01: INT;
	uAmperagemMotorGuilhotina01Sup: UINT;
	iFrequenciaMotorGuilhotina01Sup: INT;
	uAmperagemMotorGuilhotina01Inf: UINT;
	iFrequenciaMotorGuilhotina01Inf: INT;
	uAmperagemMotorGuilhotina02: UINT;
	iFrequenciaMotorGuilhotina02: INT;
	uAmperagemMotorLimpResfr02: UINT;
	iFrequenciaMotorLimpResfr02: INT;
	uAmperagemMotorCaixaForno: UINT;
	iFrequenciaMotorCaixaForno: INT;
	uAmperagemMotorVentConvec: UINT;
	iFrequenciaMotorVentConvec: INT;
	uAmperagemMotorVentConvecSai: UINT;
	iFrequenciaMotorVentConvecSai: INT;
	uAmperagemMotorVentilador01: UINT;
	iFrequenciaMotorVentilador01: INT;
	uAmperagemMotorVentilador02: UINT;
	iFrequenciaMotorVentilador02: INT;
	uAmperagemMotorVentilador03: UINT;
	iFrequenciaMotorVentilador03: INT;
	uAmperagemMotorVentilador04: UINT;
	iFrequenciaMotorVentilador04: INT;
END_VAR

(* ---- GVL_ReadStatusOnline.gvl ---- *)
VAR_GLOBAL
	/// LEITURA
	xOperacaoManual: BOOL;
	xOperacaoAutoma: BOOL;
	xOperacaoHabilitada: BOOL;
	xOperacaoStandBy: BOOL;
	xEmergencia: BOOL;
	xBtEmergenciaAcionado: BOOL;
	xResistenciasLigadas: BOOL;
	xHomeDuctosResfriadorInf01Ok: BOOL;
	xHomeDuctosResfriadorSup01Ok: BOOL;
	xHomeDuctosResfriadorInf02Ok: BOOL;
	xHomeDuctosResfriadorSup02Ok: BOOL;
	xHomeGuilhotina01Ok: BOOL;
	xHomeGuilhotina01SupOk: BOOL;
	xHomeGuilhotina01InfOk: BOOL;
	xHomeGuilhotina02Ok: BOOL;
	/// MAQUINA GERAL
	uStatusOperacao: UINT;
	uStatusInicioCiclo: UINT;
	xMaquinaEmCiclo: BOOL;
	xMaquinaEmEspera: BOOL;
	/// AQUECIMENTO
	uStatusAquecimento: INT;
	uStatusSelAquecimento: INT;
	///MESA DE ENTRADA
	uStatusMesaEntrada: UINT;
	xFimCarregamentoMesaEntrada: BOOL;
	xRetornaMesaEntrada: BOOL;
	xFimCargaMesaEntrada: BOOL;
	xFimRetornoMesaEntrada: BOOL;
	xCargaEmAutomatico: BOOL;
	///MESA DO FORNO
	uStatusMesaForno: UINT;
	iTamanhoCargaAtualForno: INT;
	iPosicaoCargaAtualForno: INT;
	iTamanhoCargaContrato: INT;
	iTamanhoCargaMaxForno: INT;
	///Variáveis de Status da Movimentação do Forno
	xFornoVazio: BOOL;
	xFornoCheio: BOOL;
	xFornoEmCiclo: BOOL;
	xFornoEmEspera: BOOL;
	xFornoFinalizando: BOOL;
	xCarregandoForno: BOOL;
	xFornoCarregado: BOOL;
	xDescarregandoForno: BOOL;
	xRetornandoForno: BOOL;
	xMesaFornoOn: BOOL;
	// MESA PASSAGEM
	xMesaPassagemOn: BOOL;
	xFimDescargaMesaPass: BOOL;
	///MESA DO RESFRIADOR
	uStatusMesaResfriador: UINT;
	iTamanhoCargaAtualResfriador: INT;
	iPosicaoCargaAtualResfriador: INT;
	///Variáveis de Status da Movimentação do Resfriador
	xResfriadorCheio: BOOL;
	xResfriadorVazio: BOOL;
	xCarregandoResfriador: BOOL;
	xResfriadorCarregado: BOOL;
	xDescarregandoResfriador: BOOL;
	xResfriadorEmCiclo: BOOL;
	xMesaResfriadorOn: BOOL;
	xPrimeiroEstagioResfriador: BOOL;
	xSegundoEstagioResfriador: BOOL;
	xTerceiroEstagioResfriador: BOOL;
	///MESA DE SAIDA
	uStatusMesaSaida: UINT;
	xInicioDescargaMesaSaida: BOOL;
	xFimDescargaMesaSaida: BOOL;
	///VENTILADOR
	///DUCTOS Inferior 01
	uStatusDuctosResfriadorInf01: INT;
	xReajustaAlturaDuctosInf01: BOOL;
	///DUCTOS Superior 01
	uStatusDuctosResfriadorSup01: INT;
	xReajustaAlturaDuctosSup01: BOOL;
	///DUCTOS Inferior 02
	uStatusDuctosResfriadorInf02: INT;
	xReajustaAlturaDuctosInf02: BOOL;
	///DUCTOS Superior 02
	uStatusDuctosResfriadorSup02: INT;
	xReajustaAlturaDuctosSup02: BOOL;
	///GUILHOTINA 01
	uStatusGuilhotina01: INT;
	///GUILHOTINA 01 SUPERIOR
	uStatusGuilhotina01Sup: INT;
	///GUILHOTINA 01 INFERIOR
	uStatusGuilhotina01Inf: INT;
	///GUILHOTINA 02
	uStatusGuilhotina02: INT;
	/// MESA BASCULANTE ENTRADA
	iStatusBasculanteEntrada: INT;
	///PRESSOSTATO
	iPressaoDaRede: INT;
	iPressaoDaMaquina: INT;
END_VAR

(* ---- GVL_Receita.gvl ---- *)
VAR_GLOBAL
	iHabilitaEscritaReceita: INT;
	iEscreverReceita: INT;
	iReceitaEscritaOk: INT;
	iReceitaEscritaFalha: INT;
	/// 1: Indica que a receita esta carregada e válida 0:Sem Receita Carregada
	xReceitaCarregadaOk: BOOL;
	sRecNomedaReceita: STRING;
	iRecEspessuraVidro: INT;
	rRecTemperaturaInferiorGeral: REAL;
	rRecTemperaturaSuperiorGeral: REAL;
	rRecPorcentagemInferiorGeral: REAL;
	rRecPorcentagemSuperiorGeral: REAL;
	rRecTemperaturaInferior: ARRAY[1..50] OF REAL;
	rRecTemperaturaSuperior: ARRAY[1..50] OF REAL;
	rRecPorcentagemInferior: ARRAY[1..50] OF REAL;
	rRecPorcentagemSuperior: ARRAY[1..50] OF REAL;
	iRecTempoDelayCarga: INT;
	iRecTempoPausaRoletes: INT;
	iRecTempoAquecimForno: INT;
	iRecTempoPosicaoForno: INT;
	///////////////
	iRecTempoVelocidadeForno: INT;
	////////////
	iRecVelocidade01Vaivem: INT;
	//////////////
	iRecVelocidade02Vaivem: INT;
	//////////////
	iRecVelocidade03Vaivem: INT;
	//////////////
	iRecVelocidadeCargaMesaForno: INT;
	///////////
	iRecVelocidadeDescargaMesaForno: INT;
	/////////
	iRecCorretorCargaMesaEntrada: INT;
	////////////
	iRecTempoPausaResistInf: INT;
	iRecTempoPausaResistSup: INT;
	iRecTempoPausa02ResistSup: INT;
	iRecTempoInicioPausa02ResistSup: INT;
	iRecTempoConveccao: INT;
	iRecTempoResfriamento: INT;
	iRecTempoTrocaEstagioResfriamento: INT;
	iRecTempoTrocaEstagio02Resfriamento: INT;
	iRecVelocidade01Ventilador01: INT;
	iRecVelocidade02Ventilador01: INT;
	iRecVelocidade03Ventilador01: INT;
	iRecVelocidadeStbVentilador01: INT;
	iRecVelocidade01Ventilador02: INT;
	iRecVelocidade02Ventilador02: INT;
	iRecVelocidade03Ventilador02: INT;
	iRecVelocidadeStbVentilador02: INT;
	iRecVelocidade01Ventilador03: INT;
	iRecVelocidade02Ventilador03: INT;
	iRecVelocidade03Ventilador03: INT;
	iRecVelocidadeStbVentilador03: INT;
	iRecVelocidade01Ventilador04: INT;
	iRecVelocidade02Ventilador04: INT;
	iRecVelocidade03Ventilador04: INT;
	iRecVelocidadeStbVentilador04: INT;
	iRecCorretorCargaMesaResfriador: INT;
	///////////
	iRecVelocidadeVaiVemResfriador: INT;
	///////////////
	iRecVelocidadeDescargaMesaResfriador: INT;
	/////////
	iRecCorretorCargaMesaSaida: INT;
	//////////////
	iRecAltura01ResfriadorInf01: INT;
	iRecAltura02ResfriadorInf01: INT;
	iRecAltura03ResfriadorInf01: INT;
	iRecAltura01ResfriadorSup01: INT;
	iRecAltura02ResfriadorSup01: INT;
	iRecAltura03ResfriadorSup01: INT;
	iRecVeneziana: INT;
	iRecPassagem: INT;
	iRecAltura01ResfriadorInf02: INT;
	iRecAltura02ResfriadorInf02: INT;
	iRecAltura03ResfriadorInf02: INT;
	iRecAltura01ResfriadorSup02: INT;
	iRecAltura02ResfriadorSup02: INT;
	iRecAltura03ResfriadorSup02: INT;
	iRecAlturaGhilhotina01: INT;
	iRecAlturaGhilhotina01Sup: INT;
	iRecAlturaGhilhotina01Inf: INT;
	iRecAlturaGhilhotina02: INT;
	iRecAjustaAlturaDuctosInf01: INT;
	iRecAjustaAlturaDuctosSup01: INT;
	iRecAjustaAlturaDuctosInf02: INT;
	iRecAjustaAlturaDuctosSup02: INT;
	iRecAjustaAlturaGuilho01: INT;
	iRecAjustaAlturaGuilho02: INT;
	dSomaReceitaSuperClp: DINT;
	iHabilitaEscritaReceitaAquec: INT;
	iReceitaAquecimEscritaOk: INT;
	/// 1: Indica que a receita esta carregada e válida 0:Sem Receita Carregada
	xReceitaAqiecimCarregadaOk: BOOL;
	iEscreverReceitaAquecim: INT;
	rRecEmissividade: REAL;
END_VAR

(* ---- GVL_Relogio.gvl ---- *)
VAR_GLOBAL
	/// Relógio em Tempo Real
	uAnoRealTime: UINT;
	uMesRealTime: UINT;
	uDiaRealTime: UINT;
	uHoraRealTime: UINT;
	uMinutoRealTime: UINT;
	uSegundoRealTime: UINT;
	uMSegundoRealTime: UINT;
	uDiaSemanaRealTime: UINT;
	uDiaAnoRealTime: UINT;
	/// Acerto do Relógio
	BtAcertaRelogioPlc: BOOL;
	uAcertoAno: UINT;
	uAcertoMes: UINT;
	uAcertoDia: UINT;
	uAcertoHora: UINT;
	uAcertoMinuto: UINT;
	uAcertoSegundo: UINT;
	uAcertoDiaSemana: UINT;
	/// Programação Horaria
	BtAtivaProgHorariaData: BOOL;
	BtAtivaProgHorariaSemana: BOOL;
	bStatusAtvProgData: BOOL;
	bStatusAtvProgSemana: BOOL;

END_VAR

(* ---- GVL_StatCanOpenDevice.gvl ---- *)
VAR_GLOBAL
	iValorCanOpenInverMesaEntraState: INT;
	iValorCanOpenInverMesaFornoState: INT;
	iValorCanOpenInverMesaPassState: INT;
	iValorCanOpenInverMesaResfrState: INT;
	iValorCanOpenInverMesaSaidaState: INT;
	iValorCanOpenInverDuctResfrSup01State: INT;
	iValorCanOpenInverDuctResfrInf01State: INT;
	iValorCanOpenInverDuctResfrSup02State: INT;
	iValorCanOpenInverDuctResfrInf02State: INT;
	iValorCanOpenInverGuilResfr01State: INT;
	iValorCanOpenInverGuilResfr02State: INT;
	iValorCanOpenInverLimpResfr02State: INT;
	iValorCanOpenInverCaixaFornoState: INT;
	iValorCanOpenInverVentila01State: INT;
	iValorCanOpenInverVentila02State: INT;
	iValorCanOpenInverVentila03State: INT;
	iValorCanOpenInverVentila04State: INT;
	iValorCanOpenInverConvecEntState: INT;
	iValorCanOpenInverConvecSaiState: INT;

	iValorCanOpenInverGuilResfr01SupState: INT;
	iValorCanOpenInverGuilResfr01InfState: INT;

	iCanOpenInverMesaEntraStateOk: BOOL;
	iCanOpenInverMesaFornoStateOk: BOOL;
	iCanOpenInverMesaPassStateOk: BOOL;
	iCanOpenInverMesaResfrStateOk: BOOL;
	iCanOpenInverMesaSaidaStateOk: BOOL;
	iCanOpenInverDuctResfrSup01StateOk: BOOL;
	iCanOpenInverDuctResfrInf01StateOk: BOOL;
	iCanOpenInverDuctResfrSup02StateOk: BOOL;
	iCanOpenInverDuctResfrInf02StateOk: BOOL;
	iCanOpenInverGuilResfr01StateOk: BOOL;
	iCanOpenInverGuilResfr02StateOk: BOOL;
	iCanOpenInverLimpResfr02StateOk: BOOL;
	iCanOpenInverCaixaFornoStateOk: BOOL;
	iCanOpenInverVentila01StateOk: BOOL;
	iCanOpenInverVentila02StateOk: BOOL;
	iCanOpenInverVentila03StateOk: BOOL;
	iCanOpenInverVentila04StateOk: BOOL;
	iCanOpenInverConvecEntStateOk: BOOL;
	iCanOpenInverConvecSaiStateOk: BOOL;

	iCanOpenInverGuilResfr01SupStateOk: BOOL;
	iCanOpenInverGuilResfr01InfStateOk: BOOL;

	xAlarmeCofInverMesaEntra: BOOL;
	xAlarmeCofInverMesaForno: BOOL;
	xAlarmeCofInverMesaPass: BOOL;
	xAlarmeCofInverMesaResfr: BOOL;
	xAlarmeCofInverMesaSaida: BOOL;
	xAlarmeCofInverResfrSup01: BOOL;
	xAlarmeCofInverResfrInf01: BOOL;
	xAlarmeCofInverResfrSup02: BOOL;
	xAlarmeCofInverResfrInf02: BOOL;
	xAlarmeCofInverGuilho01: BOOL;
	xAlarmeCofInverGuilho02: BOOL;
	xAlarmeCofInverConvecEnt: BOOL; //Superior
	xAlarmeCofInverConvecSai: BOOL; //Inferior
	xAlarmeCofInverVentila03: BOOL;

	xAlarmeCofInverGuilho01Sup: BOOL;
	xAlarmeCofInverGuilho01Inf: BOOL;
	xAlarmeCofInverCaixaForno: BOOL;

END_VAR

(* ---- GVL_StatModTcpDevice.gvl ---- *)
VAR_GLOBAL
// Global Status Modbus TCP  IOScaner valores (Não Configurado-1, Stop-3, Operacional-2).
ModbusTCP_IOScanner_Gstatus: UINT;
// Health Bit dos canais de escrita e leitura das remotas TM3BCEIP
TM3BC_ModbusTCP_1_Hb_Ch0 : BOOL;
TM3BC_ModbusTCP_1_Hb_Ch1 : BOOL;
TM3BC_ModbusTCP_2_Hb_Ch2 : BOOL;
TM3BC_ModbusTCP_2_Hb_Ch3 : BOOL;
TM3BC_ModbusTCP_3_Hb_Ch4 : BOOL;
TM3BC_ModbusTCP_3_Hb_Ch5 : BOOL;
TM3BC_ModbusTCP_4_Hb_Ch6 : BOOL;
TM3BC_ModbusTCP_4_Hb_Ch7 : BOOL;
// Habilitação dos canais de escrita e leitura das remotas TM3BCEIP
TM3BC_ModbusTCP_1_En_Ch0 : BOOL;
TM3BC_ModbusTCP_1_En_Ch1 : BOOL;
TM3BC_ModbusTCP_2_En_Ch2 : BOOL;
TM3BC_ModbusTCP_2_En_Ch3 : BOOL;
TM3BC_ModbusTCP_3_En_Ch4 : BOOL;
TM3BC_ModbusTCP_3_En_Ch5 : BOOL;
TM3BC_ModbusTCP_4_En_Ch6 : BOOL;
TM3BC_ModbusTCP_4_En_Ch7 : BOOL;

END_VAR

(* ---- GVL_SuperClp.gvl ---- *)
VAR_GLOBAL
	/// Parametros Buffer 01
	/// Parametros do Forno
	rBufferSetTemperaturaInferiorGeral: REAL;
	rBufferSetTemperaturaSuperiorGeral: REAL;
	rBufferSetPorcentagemInferiorGeral: REAL;
	rBufferSetPorcentagemSuperiorGeral: REAL;
	rBufferSetTemperaturaInferior: ARRAY[1..60] OF REAL;
	rBufferSetTemperaturaSuperior: ARRAY[1..60] OF REAL;
	rBufferSetPorcentagemInferior: ARRAY[1..60] OF REAL;
	rBufferSetPorcentagemSuperior: ARRAY[1..60] OF REAL;
	iBufferTempoPausaResistInf: INT;
	iBufferTempoPausaResistSup: INT;
	iBufferTempoPausa02ResistSup: INT;
	iBufferTempoInicioPausa02ResistSup: INT;
	iBufferTempoConveccao: INT;
	iBufferTempoDelayCarga: INT;
	iBufferTempoPausaRoletes: INT;
	iBufferTempoAquecimForno: INT;
	iBufferTempoPosicaoForno: INT;
	iBufferTempoVelocidadeForno: INT;
	iBufferVelocidade01Vaivem: INT;
	iBufferVelocidade02Vaivem: INT;
	iBufferVelocidade03Vaivem: INT;
	iBufferVelocidadeCargaMesadoForno: INT;
	iBufferVelocidadeDescargaMesadoForno: INT;
	iBufferCorretorCargaMesaEntrada: INT;
	///Parametros do Resfriamento
	iBufferTempoResfriamento: INT;
	iBufferValAltura01ResfriadorInf01: INT;
	iBufferValAltura02ResfriadorInf01: INT;
	iBufferValAltura03ResfriadorInf01: INT;
	iBufferValAltura01ResfriadorSup01: INT;
	iBufferValAltura02ResfriadorSup01: INT;
	iBufferValAltura03ResfriadorSup01: INT;
	iBufferValAltura01ResfriadorInf02: INT;
	iBufferValAltura02ResfriadorInf02: INT;
	iBufferValAltura03ResfriadorInf02: INT;
	iBufferValAltura01ResfriadorSup02: INT;
	iBufferValAltura02ResfriadorSup02: INT;
	iBufferValAltura03ResfriadorSup02: INT;
	iBufferAlturaGhilhotina01: INT;
	iBufferAlturaGhilhotina01Sup: INT;
	iBufferAlturaGhilhotina01Inf: INT;
	iBufferAlturaGhilhotina02: INT;
	iBufferVelocidade01Ventilador01: INT;
	iBufferVelocidade02Ventilador01: INT;
	iBufferVelocidade03Ventilador01: INT;
	iBufferVelocidade01Ventilador02: INT;
	iBufferVelocidade02Ventilador02: INT;
	iBufferVelocidade03Ventilador02: INT;
	iBufferVelocidade01Ventilador03: INT;
	iBufferVelocidade02Ventilador03: INT;
	iBufferVelocidade03Ventilador03: INT;
	iBufferVelocidade01Ventilador04: INT;
	iBufferVelocidade02Ventilador04: INT;
	iBufferVelocidade03Ventilador04: INT;
	iBufferTempoTrocaEstagioResfriamento: INT;
	iBufferTempoTrocaEstagio02Resfriamento: INT;
	iBufferCorretorCargaMesaResfriador: INT;
	iBufferVelocidadeVaiVemResfriador: INT;
	iBufferVelocidadeDescargaMesadoResfriador: INT;
	iBufferCorretorCargaMesaSaida: INT;
	iBufferVeneziana: INT;
	iBufferPassagem: INT;
	rBufferEmissividade	: REAL;
	/// Parametros Buffer 02
	///Parametros do Resfriamento
	iBuffer02TempoResfriamento: INT;
	iBuffer02ValAltura01ResfriadorInf01: INT;
	iBuffer02ValAltura02ResfriadorInf01: INT;
	iBuffer02ValAltura03ResfriadorInf01: INT;
	iBuffer02ValAltura01ResfriadorSup01: INT;
	iBuffer02ValAltura02ResfriadorSup01: INT;
	iBuffer02ValAltura03ResfriadorSup01: INT;
	iBuffer02ValAltura01ResfriadorInf02: INT;
	iBuffer02ValAltura02ResfriadorInf02: INT;
	iBuffer02ValAltura03ResfriadorInf02: INT;
	iBuffer02ValAltura01ResfriadorSup02: INT;
	iBuffer02ValAltura02ResfriadorSup02: INT;
	iBuffer02ValAltura03ResfriadorSup02: INT;
	iBuffer02AlturaGhilhotina01: INT;
	iBuffer02AlturaGhilhotina01Sup: INT;
	iBuffer02AlturaGhilhotina01Inf: INT;
	iBuffer02AlturaGhilhotina02: INT;
	iBuffer02Velocidade01Ventilador01: INT;
	iBuffer02Velocidade02Ventilador01: INT;
	iBuffer02Velocidade03Ventilador01: INT;
	iBuffer02Velocidade01Ventilador02: INT;
	iBuffer02Velocidade02Ventilador02: INT;
	iBuffer02Velocidade03Ventilador02: INT;
	iBuffer02Velocidade01Ventilador03: INT;
	iBuffer02Velocidade02Ventilador03: INT;
	iBuffer02Velocidade03Ventilador03: INT;
	iBuffer02Velocidade01Ventilador04: INT;
	iBuffer02Velocidade02Ventilador04: INT;
	iBuffer02Velocidade03Ventilador04: INT;
	iBuffer02TempoTrocaEstagioResfriamento: INT;
	iBuffer02TempoTrocaEstagio02Resfriamento: INT;
	iBuffer02CorretorCargaMesaResfriador: INT;
	iBuffer02VelocidadeVaiVemResfriador: INT;
	iBuffer02VelocidadeDescargaMesadoResfriador: INT;
	iBuffer02CorretorCargaMesaSaida: INT;
	iBuffer02Veneziana: INT;
	iBuffer02Passagem: INT;
	rBuffer02Emissividade:REAL;
	/// ESCRITA - LEITURA
	///Parâmetros On-line
	/// Parâmetros Forno pós Buffer01
	rSetTemperaturaInferiorGeral: REAL;
	rSetTemperaturaSuperiorGeral: REAL;
	rSetPorcentagemInferiorGeral: REAL;
	rSetPorcentagemSuperiorGeral: REAL;
	rSetTemperaturaInferior: ARRAY[1..60] OF REAL;
	rSetTemperaturaSuperior: ARRAY[1..60] OF REAL;
	rSetPorcentagemInferior: ARRAY[1..60] OF REAL;
	rSetPorcentagemSuperior: ARRAY[1..60] OF REAL;
	iTempoPausaResistInf: INT;
	iTempoPausaResistSup: INT;
	iTempoPausa02ResistSup: INT;
	iTempoInicioPausa02ResistSup: INT;
	iTempoConveccao: INT;
	iTempoDelayCarga: INT;
	iTempoPausaRoletes: INT;
	iTempoAquecimForno: INT;
	iTempoPosicaoForno: INT;
	iTempoVelocidadeForno: INT;
	iVelocidade01Vaivem: INT;
	iVelocidade02Vaivem: INT;
	iVelocidade03Vaivem: INT;
	iVelocidadeCargaMesadoForno: INT;
	iVelocidadeDescargaMesadoForno: INT;

	/// Parâmetros Resfriamento
	/// Parametros Resfriamento pós Buffer 02
	iTempoResfriamento: INT;
	iValAltura01ResfriadorInf01: INT;
	iValAltura02ResfriadorInf01: INT;
	iValAltura03ResfriadorInf01: INT;
	iValAltura01ResfriadorSup01: INT;
	iValAltura02ResfriadorSup01: INT;
	iValAltura03ResfriadorSup01: INT;
	iValAltura01ResfriadorInf02: INT;
	iValAltura02ResfriadorInf02: INT;
	iValAltura03ResfriadorInf02: INT;
	iValAltura01ResfriadorSup02: INT;
	iValAltura02ResfriadorSup02: INT;
	iValAltura03ResfriadorSup02: INT;
	iAlturaGhilhotina01: INT;
	iAlturaGhilhotina01Sup: INT;
	iAlturaGhilhotina01Inf: INT;
	iAlturaGhilhotina02: INT;
	iVelocidade01Ventilador01: INT;
	iVelocidade02Ventilador01: INT;
	iVelocidade03Ventilador01: INT;
	iVelocidade01Ventilador02: INT;
	iVelocidade02Ventilador02: INT;
	iVelocidade03Ventilador02: INT;
	iVelocidade01Ventilador03: INT;
	iVelocidade02Ventilador03: INT;
	iVelocidade03Ventilador03: INT;
	iVelocidade01Ventilador04: INT;
	iVelocidade02Ventilador04: INT;
	iVelocidade03Ventilador04: INT;
	iTempoTrocaEstagioResfriamento: INT;
	iTempoTrocaEstagio02Resfriamento: INT;

	iVelocidadeVaiVemResfriador: INT;
	iVelocidadeDescargaMesadoResfriador: INT;

	iVeneziana: INT;
	iPassagem: INT;
	BtParamMesaForno: BOOL;
	BtParamMesaResfriador: BOOL;
	BtParamDuctosResfriadorInf01: BOOL;
	BtParamDuctosResfriadorSup01: BOOL;
	BtParamDuctosResfriadorInf02: BOOL;
	BtParamDuctosResfriadorSup02: BOOL;
	BtParamGuilhotina01: BOOL;
	BtParamGuilhotina01Sup: BOOL;
	BtParamGuilhotina01Inf: BOOL;
	BtParamGuilhotina02: BOOL;
	xIniciaHomeDuctosInf01: BOOL;
	xIniciaHomeDuctosSup01: BOOL;
	xIniciaHomeDuctosInf02: BOOL;
	xIniciaHomeDuctosSup02: BOOL;
	xIniciaHomeGuilhotina01: BOOL;
	xIniciaHomeGuilhotina01Sup: BOOL;
	xIniciaHomeGuilhotina01Inf: BOOL;
	xIniciaHomeGuilhotina02: BOOL;
	BtHabDesabBloqueio: BOOL;
	BtDesbloqueio: BOOL;
	BtAbreVeneziana: BOOL;
	BtFechaVeneziana: BOOL;
	BtAbreVenezVentInfPass: BOOL;
	BtFechVenezVentInfPass: BOOL;
	BtHabilitaResistenciasGeralInferior: BOOL;
	BtDesabilitaResistenciasGeralInferior: BOOL;
	BtHabilitaResistenciasGeralSuperior: BOOL;
	BtDesabilitaResistenciasGeralSuperior: BOOL;
	BtHabilitaResistenciaInferior: ARRAY[1..60] OF BOOL;
	BtHabilitaResistenciaSuperior: ARRAY[1..60] OF BOOL;
	BtHabDesabResistConveccaoEnt: BOOL;
	BtHabDesabResistConveccaoSai: BOOL;
	bIniciaTesteResistencias: BOOL;
	bAbortaTesteResistencias: BOOL;
	bResetTesteResistencias: BOOL;
	BtForceResistenciaInferior: ARRAY[1..60] OF BOOL;
	BtForceResistenciaSuperior: ARRAY[1..60] OF BOOL;
	BtTesteResistencias: BOOL;
	BtTesteResistenciaAutomatico: BOOL;
	BtTesteResistenciaManual: BOOL;
	BtTesteEntradaSaidas: BOOL;
	BtSelecaoTermopares: BOOL;
	BtResetAlarmesGerais: BOOL;
	BtRestart: BOOL;
	BtAbortaStandByCiclo: BOOL;
	xBtHabIncremento: BOOL;
	xBtIniciaTesteNobreak: BOOL;

	rEmissividade	: REAL;
END_VAR

(* ---- GVL_Velocidades.gvl ---- *)
VAR_GLOBAL
	///Velocidade Sem corretor
	iVelCargaMesaEntradaVidroFin: INT;
	///Velodidade Aplicada Com Corretor
	iVelCargaMeEntradaVidroFin: INT;
	///Velocidade Sem corretor
	iVelCargaMesaEntrada: INT;
	///Velodidade Aplicada Com Corretor
	iVelCargaMeEntrada: INT;
	///Comum
	iVelRetornoMesaEntrada: INT;
	///Velocidade Sem corretor
	iVelCargaResfriadorVidroFin: INT;
	///Velodidade Aplicada Com Corretor
	iVelCargaMeResfriadorVidroFin: INT;
	///Velocidade Sem corretor
	iVelCargaResfriador: INT;
	///Velodidade Aplicada Com Corretor
	iVelCargaMeResfriador: INT;
	///Velocidade Sem corretor
	iVelCargaMesaSaidaVidroFin: INT;
	///Velodidade Aplicada Com Corretor
	iVelCargaMeSaidaVidroFin: INT;
	///Velocidade Sem corretor
	iVelCargaMesaSaida: INT;
	///Velodidade Aplicada Com Corretor
	iVelCargaMeSaida: INT;
END_VAR

(* ---- GVL_WriteComandos.gvl ---- *)
VAR_GLOBAL
	xAbortaCicloForno: BOOL;
	xBtHmiIniciaCiclo: BOOL;
	xBtHmiFinalizaCiclo: BOOL;
	xBtSairForno: BOOL;
	xBtSairResfriamento: BOOL;
	xBtAbortaCiclo: BOOL;
	xBtAbrePortaEntradaForno: BOOL;
	xBtAbrePortaSaidaForno: BOOL;
	xBtForceConveccao: BOOL;
	xBtSobeGuilhtina01Manual: BOOL;
	xBtDesceGuilhotina01Manual: BOOL;
	xBtSobeGuilhtina02Manual: BOOL;
	xBtDesceGuilhotina02Manual: BOOL;
	xBtSobeForno: BOOL;
	xBtDesceForno: BOOL;
	xBtLigaVentiPainelManual: BOOL;
	xBtDuctosInf01Enable: BOOL;
	xBtDuctosSup01Enable: BOOL;
	xBtDuctosInf02Enable: BOOL;
	xBtDuctosSup02Enable: BOOL;
	xBtGuilhotina01Enable: BOOL;
	xBtGuilhotina01SupEnable: BOOL;
	xBtGuilhotina01InfEnable: BOOL;
	xBtGuilhotina02Enable: BOOL;
	xBtLigaAquecimentoRampa: BOOL;
	xBtLigaAquecimento: BOOL;
	xBtDesligaAquecimento: BOOL;
	xBtSelAqueceRampaReceita: BOOL;
	xBtSelAqueceRapidoLento: BOOL;
END_VAR
